# B&R Automation Studio project RobotNewEra (part 11)

#### iolist.c
```c
/************************************************************************************************************************/
/* Object name: iolist.c																								*/
/* Author:      Andreas Hager, B&R																						*/
/* Site:        Eggelsberg                                                                                            	*/
/* Created:     24-Feb-2006                                                                                           	*/
/* Restriction: 													      		                                      	*/
/* Description: Function to read out configured IO data points                                                      	*/
/*----------------------------------------------------------------------------------------------------------------------*/
/* Version 1.00			24-Feb-2006		 Andreas Hager			Official release								  		*/
/*----------------------------------------------------------------------------------------------------------------------*/
/* Version 1.01			13-Dec-2006		 Andreas Hager			Comment added									  		*/
/*----------------------------------------------------------------------------------------------------------------------*/
/* Version 2.00			16-Jul-2008		 Andreas Hager			AS3 - Changes for GCC 4.1.1								*/
/*----------------------------------------------------------------------------------------------------------------------*/
/* Version 2.01			16-Sep-2009		 Andreas Hager			Bugfix for memset in StringParser()						*/
/*----------------------------------------------------------------------------------------------------------------------*/
/* Development tool: B&R Automation Studio V3.0.71.31 SP05 																*/
/*----------------------------------------------------------------------------------------------------------------------*/
/* Comment:                                                                                                           	*/
/************************************************************************************************************************/

#include <ModDiag.h>
#include <bur/plctypes.h>
#include <AsIOMMan.h>
#include <DataObj.h>
#include <string.h>
#include <AsIODiag.h>
#include <Sys_lib.h>
#include <Standard.h>
#include "internal_h.h"

#define	CREATE_HW_INFO		0
#define	ALLOC_MEMORY		1
#define	GET_MODULE_NAME		2
#define	GET_MODULE_PATH		3
#define	CHECK_NEXT_MODULE	4
#define	DISPOSE_INFO		5

#define	MAX_LENGTH			512

#define	PV_NAME_OVERFLOW	50001
#define	FUNCTION_BUSY		65535

static	AsIOMMCopy_typ		IOMapCopy;
static	DatObjDelete_typ	DataModuleDelete;
static	DatObjInfo_typ		DataModuleInfo;

/* Function to get io module information */
unsigned short ModulesInformation(UDINT pModuleInfo);
/* Function to parse iomap data */
unsigned short StringParser(UDINT pBuffer, UDINT pIOData, UDINT pIOCounter, USINT Option);
/* Function to sort io list depending on device */
void SortIOList(UDINT pIOList, UINT IOEntries);

unsigned short IOList(unsigned long pIOInformation)
{	USINT	*Parser = 0, NumberConfiguredModules = 0;
	UINT	xcnt = 0, ycnt  = 0, TotalIOs = 0, OldDigitalInputs = 0, OldDigitalOutputs = 0, OldAnalogInputs = 0, OldAnalogOutputs = 0, DPIndex = 0,
			ModuleStatus = 0, ParserStatus = 0, AllocStatus = 0, StatusFree = 0;
	UDINT	MaxAdr = 0;
	STRING	ParserString[800];

	IODPList_typ			*IOList = 0;
	SingleModuleInfo_typ	*SingleModuleInfo = 0;
	SingleIOEntry_typ		*SingleIOEntry = 0;
	IOStringInfo_typ		EntryInfo;
	IOCounter_typ			IOCounter;
	ModuleInfo_typ			ModuleInformation;

	memset(&(EntryInfo), 0, sizeof(EntryInfo));
	memset(&(ModuleInformation), 0, sizeof(ModuleInformation));
	memset(&(IOCounter), 0, sizeof(IOCounter));

	*(UDINT*)&IOList = pIOInformation;

	/* Get module information */
	do
	{	ModuleStatus = ModulesInformation((UDINT)&(ModuleInformation));
	} while(ModuleStatus == 65535);

	if(ModuleStatus)
	{	return(ModuleStatus);
	}

	/* Number of configured modules */
	NumberConfiguredModules = ModuleInformation.TotalModules - ModuleInformation.IgnoredModules;

	/* Pointer to module information buffer */
	*(UDINT*)&SingleModuleInfo = ModuleInformation.StartAdrBuffer;

	/* Check if io data module already exists */
	DataModuleInfo.enable = 1;
	DataModuleInfo.pName = (UDINT)"iomap_io";
	DatObjInfo(&DataModuleInfo);

	if(DataModuleInfo.status == 0)
	{	DataModuleDelete.enable = 1;
		DataModuleDelete.ident = DataModuleInfo.ident;
		DatObjDelete(&DataModuleDelete);
	}

	/* Generate data module of iomap file */
	do
	{	IOMapCopy.enable = 1;
		IOMapCopy.pModuleName = (UDINT)"iomap";
		IOMapCopy.pNewModule = (UDINT)"iomap_io";
		IOMapCopy.memType = 65;
		AsIOMMCopy(&IOMapCopy);
	} while(IOMapCopy.status == 65535);

	if(IOMapCopy.status)
	{	return(IOMapCopy.status);
	}

	DataModuleInfo.enable = 1;
	DataModuleInfo.pName = (UDINT)"iomap_io";
	DatObjInfo(&DataModuleInfo);

	if(DataModuleInfo.status)
	{	return(DataModuleInfo.status);
	}

	MaxAdr = DataModuleInfo.pDatObjMem + DataModuleInfo.len;

	/* Pointer to the start address of io data module */
	*(UDINT*)&Parser = DataModuleInfo.pDatObjMem;

	while((UDINT)Parser < MaxAdr)
	{
		/* Each line with information starts with <LN */
		if(!memcmp((UDINT*)Parser, "<LN ", 4))
		{	Parser = Parser + 4;

			/* Copy data tiil </LN> */
			for(xcnt = 0; xcnt < 800; xcnt++)
			{	if(!memcmp((UDINT*)Parser, "</LN>", 5))
				{	ParserString[xcnt] = 0;
					Parser = Parser + 5;

					/* Check string for information --> Option = 0 - check number of completed entries */
					ParserStatus = StringParser((UDINT)&(ParserString), (UDINT)&(EntryInfo), (UDINT)&(IOCounter), 0);

					if(ParserStatus)
						return(ParserStatus);

					memset(&(ParserString), 0, sizeof(ParserString));
					break;
				}
				else
				{	ParserString[xcnt] = *Parser;
					Parser++;
				}
			}
		}
		/* Increase pointer */
		else
		{	Parser++;
		}
	}

	TotalIOs = IOCounter.NumberDigitalInputs + IOCounter.NumberDigitalOutputs + IOCounter.NumberAnalogInputs + IOCounter.NumberAnalogOutputs;

	if(TotalIOs == 0)
		return(0);

	/* Allocate memory */
	do
	{	AllocStatus = TMP_alloc(sizeof(SingleIOEntry_typ)*TotalIOs, (void*)&(IOList->StartAdrBuffer));
	} while(AllocStatus == 65535);

	if(AllocStatus)
	{	return(AllocStatus);
	}

	/* Pare data module again */
	memset((void*)IOList->StartAdrBuffer, 0, sizeof(SingleIOEntry_typ)*TotalIOs);
	*(UDINT*)&SingleIOEntry = IOList->StartAdrBuffer;
	memset(&(IOCounter), 0, sizeof(IOCounter));
	memset(&(ParserString), 0, sizeof(ParserString));

	*(UDINT*)&Parser = DataModuleInfo.pDatObjMem;

	while((UDINT)Parser < MaxAdr)
	{
		/* Each line with information starts with <LN */
		if(!memcmp((UDINT*)Parser, "<LN ", 4))
		{	Parser = Parser + 4;

			/* Copy data tiil </LN> */
			for(xcnt = 0; xcnt < 800; xcnt++)
			{	if(!memcmp((UDINT*)Parser, "</LN>", 5))
				{	ParserString[xcnt] = 0;
					Parser = Parser + 5;

					/* Check string for information --> Option = 1 - copy information to EntryInfo */
					ParserStatus = StringParser((UDINT)&(ParserString), (UDINT)&(EntryInfo), (UDINT)&(IOCounter), 1);

					if(ParserStatus)
						return(ParserStatus);

					/* Copy information from EntryInfo to allocated buffer */
					if(OldDigitalInputs != IOCounter.NumberDigitalInputs || OldDigitalOutputs != IOCounter.NumberDigitalOutputs ||
						OldAnalogInputs != IOCounter.NumberAnalogInputs || OldAnalogOutputs != IOCounter.NumberAnalogOutputs)
					{	strcpy((SingleIOEntry + DPIndex)->Device, EntryInfo.Device);
						strcpy((SingleIOEntry + DPIndex)->ID, EntryInfo.ID);
						strcpy((SingleIOEntry + DPIndex)->LogicalName, EntryInfo.LogicalName);
						(SingleIOEntry + DPIndex)->Type = EntryInfo.Type;
						strcpy((SingleIOEntry + DPIndex)->PVName, EntryInfo.PVName);

						memset(&(EntryInfo), 0, sizeof(EntryInfo));

						/* Copy information about io module */
						for(ycnt = 0; ycnt < NumberConfiguredModules; ycnt++)
						{	if(!strcmp((SingleIOEntry + DPIndex)->Device, (SingleModuleInfo + ycnt)->ModulePath))
							{	strcpy((SingleIOEntry + DPIndex)->ModuleName, (SingleModuleInfo + ycnt)->ModuleName);
								break;
							}
						}
						OldDigitalInputs = IOCounter.NumberDigitalInputs;
						OldDigitalOutputs = IOCounter.NumberDigitalOutputs;
						OldAnalogInputs = IOCounter.NumberAnalogInputs;
						OldAnalogOutputs = IOCounter.NumberAnalogOutputs;

						DPIndex++;
					}
					memset(&(ParserString), 0, sizeof(ParserString));
					break;
				}
				else
				{	ParserString[xcnt] = *Parser;
					Parser++;
				}
			}
		}
		else
		{	Parser++;
		}
	}

	/* Free memory with io module information */
	StatusFree = TMP_free(sizeof(SingleModuleInfo_typ)*ModuleInformation.TotalModules, (void*)ModuleInformation.StartAdrBuffer);

	if(StatusFree)
	{	return(StatusFree);
	}

	/* Sort io list */
	SortIOList(IOList->StartAdrBuffer, TotalIOs);

	/* Copy number of ios */
	IOList->NumberDigitalInput = IOCounter.NumberDigitalInputs;
	IOList->NumberDigitalOutput = IOCounter.NumberDigitalOutputs;
	IOList->NumberAnalogInput = IOCounter.NumberAnalogInputs;
	IOList->NumberAnalogOutput = IOCounter.NumberAnalogOutputs;
	IOList->TotalIONumber = IOCounter.NumberDigitalInputs + IOCounter.NumberDigitalOutputs + IOCounter.NumberAnalogInputs + IOCounter.NumberAnalogOutputs;
	return(0);
}

/* Function to get io module information */
unsigned short ModulesInformation(UDINT pModuleInfo)
{	static	DiagCreateInfo_typ		CreateHWInfo;
	static	DiagGetStrInfo_typ		GetModulePath, GetModuleName;
	static	DiagDisposeInfo_typ		DisposeInfo;
	static	SingleModuleInfo_typ	*SingleModuleInfo = 0;

	USINT	*pUSINT1 = 0, *pUSINT2 = 0;
	UINT	Status = 0;
	STRING	ModulePath[40], ModuleName[20];

	ModuleInfo_typ			*ModuleInfo = 0;

	memset(&(ModulePath), 0, sizeof(ModulePath));
	memset(&(ModuleName), 0, sizeof(ModuleName));

	*(UDINT*)&ModuleInfo = pModuleInfo;

	switch(ModuleInfo->Step)
	{
		/* Get information about configured hardware */
		case CREATE_HW_INFO:
			CreateHWInfo.enable = 1;
			CreateHWInfo.infoKind = asdiagCONFIGURED;

			DiagCreateInfo(&CreateHWInfo);
			Status = CreateHWInfo.status;

			if(CreateHWInfo.status == 0)
			{	ModuleInfo->TotalModules = CreateHWInfo.nrEntries;
				ModuleInfo->HWIdent = CreateHWInfo.ident;
				ModuleInfo->Step = ALLOC_MEMORY;
				Status = FUNCTION_BUSY;
			}
		break;

		/* Allocate memory for hardware information depending on number of modules */
		case ALLOC_MEMORY:
			Status = TMP_alloc(sizeof(SingleModuleInfo_typ)*ModuleInfo->TotalModules, (void*)&(ModuleInfo->StartAdrBuffer));

			if(Status == 0)
			{	memset((void*)ModuleInfo->StartAdrBuffer, 0, sizeof(SingleModuleInfo_typ)*ModuleInfo->TotalModules);
				*(UDINT*)&SingleModuleInfo = ModuleInfo->StartAdrBuffer;
				/* Set module index on next module after panel */
				ModuleInfo->ModuleIndex = 1;
				ModuleInfo->IgnoredModules = 1;
				ModuleInfo->Step = GET_MODULE_NAME;
				Status = FUNCTION_BUSY;
			}
		break;

		/* Get name for each hardware module */
		case GET_MODULE_NAME:
			GetModuleName.enable = 1;
			GetModuleName.ident = CreateHWInfo.ident;
			GetModuleName.index = ModuleInfo->ModuleIndex;
			GetModuleName.infoCode = asdiagCONFIG_MODULE;
			GetModuleName.pBuffer = (UDINT)ModuleName;
			GetModuleName.bufferLen = sizeof(ModuleName);

			DiagGetStrInfo(&GetModuleName);
			Status = GetModuleName.status;

			if(GetModuleName.status == 0)
			{	*(UDINT*)&pUSINT1 = (UDINT)(ModuleName + 1);
				*(UDINT*)&pUSINT2 = (UDINT)(ModuleName + 2);

				/* Ignore IF and ACxxx */
				if((*pUSINT1 == 'I' && *pUSINT2 == 'F') || (*pUSINT1 == 'A' && *pUSINT2 == 'C'))
				{	ModuleInfo->IgnoredModules++;
					ModuleInfo->Step = CHECK_NEXT_MODULE;
				}
				else
				{	strcpy((SingleModuleInfo + (ModuleInfo->ModuleIndex - ModuleInfo->IgnoredModules))->ModuleName, ModuleName);
					ModuleInfo->Step = GET_MODULE_PATH;
				}
				Status = FUNCTION_BUSY;
			}
		break;

		/* Get path for each hardware module */
		case GET_MODULE_PATH:
			GetModulePath.enable = 1;
			GetModulePath.ident = CreateHWInfo.ident;
			GetModulePath.index = ModuleInfo->ModuleIndex;
			GetModulePath.infoCode = asdiagPATH;
			GetModulePath.pBuffer = (UDINT)ModulePath;
			GetModulePath.bufferLen = sizeof(ModulePath);

			DiagGetStrInfo(&GetModulePath);
			Status = GetModulePath.status;

			if(GetModulePath.status == 0)
			{	strcpy((SingleModuleInfo + (ModuleInfo->ModuleIndex - ModuleInfo->IgnoredModules))->ModulePath, ModulePath);
				ModuleInfo->Step = CHECK_NEXT_MODULE;
				Status = FUNCTION_BUSY;
			}
		break;

		/* Select nex module */
		case CHECK_NEXT_MODULE:
			if(ModuleInfo->ModuleIndex < ModuleInfo->TotalModules - 1)
			{	ModuleInfo->ModuleIndex++;
				ModuleInfo->Step = GET_MODULE_NAME;
			}
			else
			{	ModuleInfo->Step = DISPOSE_INFO;
			}
			Status = FUNCTION_BUSY;
		break;

		/* Dispose information */
		case DISPOSE_INFO:
			DisposeInfo.enable = 1;
			DisposeInfo.ident = ModuleInfo->HWIdent;

			DiagDisposeInfo(&DisposeInfo);

			if(DisposeInfo.status == 0)
			{	ModuleInfo->Step = CREATE_HW_INFO;
			}
		break;
	}
	return(Status);
}

/* Function to parse iomap data */
unsigned short StringParser(UDINT pBuffer, UDINT pIOData, UDINT pIOCounter, USINT Option)
{	USINT	*Parser = 0, Element = 0;
	UINT xcnt = 0;
	STRING	Data[MAX_LENGTH], ID[60], Type[40], DType[40], Device1[60], DPName1[34], Kind1[40], Device2[60], DPName2[34], Kind2[40];

	IOStringInfo_typ	*EntryInfo = 0;
	IOCounter_typ		*IOCounter = 0;

	memset(&(Data), 0, sizeof(Data));
	memset(&(ID), 0, sizeof(ID));
	memset(&(Type), 0, sizeof(Type));
	memset(&(DType), 0, sizeof(DType));
	memset(&(Device1), 0, sizeof(Device1));
	memset(&(DPName1), 0, sizeof(DPName1));
	memset(&(Kind1), 0, sizeof(Kind1));
	memset(&(Device2), 0, sizeof(Device2));
	memset(&(DPName2), 0, sizeof(DPName2));
	memset(&(Kind2), 0, sizeof(Kind2));

	*(UDINT*)&Parser = pBuffer;
	*(UDINT*)&EntryInfo = pIOData;
	*(UDINT*)&IOCounter = pIOCounter;

	while(*Parser)
	{	/* Information starts with " */
		while(*Parser != '"' && *Parser)
		{	Parser++;
		}
		if(!*Parser)
			break;
		else
			Parser++;

		/* Information ends with " */
		while(*Parser != '"' && *Parser)
		{	Data[xcnt] = *Parser;
			Parser++;
			xcnt++;
			if(xcnt == MAX_LENGTH)
				return(PV_NAME_OVERFLOW);
		}
		Parser++;
		Data[xcnt] = 0;
		xcnt = 0;

		/* Element 0 --> IO ID */
		if(Element == 0)
		{	strcpy(ID, Data);
			memcpy(Type, Data, 3);
		}
		/* Element 1 --> Data type */
		else if(Element == 1)
		{	strcpy(DType, Data);
		}
		/* Element 2 --> Device */
		else if(Element == 2)
		{	strcpy(Device1, Data);
		}
		/* Element 3 --> Data point name */
		else if(Element == 3)
		{	strcpy(DPName1, Data);
		}
		/* Element 4 --> Kind */
		else if(Element == 4)
		{	strcpy(Kind1, Data);
		}
		/* Element 5 --> Device */
		else if(Element == 5)
		{	strcpy(Device2, Data);
		}
		/* Element 6 --> Data point name */
		else if(Element == 6)
		{	strcpy(DPName2, Data);
		}
		/* Elemtn 7 --> Kind */
		else if(Element == 7)
		{	strcpy(Kind2, Data);
		}

		Element++;
		memset(&(Data), 0, sizeof(Data));
	}

	/* If less than 8 elements are detected --> information is completed */
	if(Element != 8)
	{	Element = 0;
		return(0);
	}

	/* Type %IX --> Digital input */
	if(Element == 8 && !strcmp(Type, "%IX"))
	{	IOCounter->NumberDigitalInputs++;
	}
	/* Type %QX --> Digital output */
	else if(Element == 8 && !strcmp(Type, "%QX"))
	{	IOCounter->NumberDigitalOutputs++;
	}
	/* Type %IW --> Analog input */
	else if(Element == 8 && !strcmp(Type, "%IW"))
	{	IOCounter->NumberAnalogInputs++;
	}
	/* Type %QW --> Analog output */
	else if(Element == 8 && !strcmp(Type, "%QW"))
	{	IOCounter->NumberAnalogOutputs++;
	}

	/* If option = 1 --> copy all information to EntryInfo */
	if(Option == 1 && Element == 8)
	{	strcpy(EntryInfo->ID, ID);

		if(!strcmp(Type, "%IX"))
		{	EntryInfo->Type = 1;
			if(!strcmp(Kind1, "io"))
			{	strcpy(EntryInfo->LogicalName, DPName1);
			}
			else if(!strcmp(Kind2, "io"))
			{	strcpy(EntryInfo->LogicalName, DPName2);
			}
		}
		else if(!strcmp(Type, "%QX"))
		{	EntryInfo->Type = 2;
			if(!strcmp(Kind1, "io"))
			{	strcpy(EntryInfo->LogicalName, DPName1);
			}
			else if(!strcmp(Kind2, "io"))
			{	strcpy(EntryInfo->LogicalName, DPName2);
			}
		}
		else if(!strcmp(Type, "%IW"))
		{	EntryInfo->Type = 3;
			if(!strcmp(Kind1, "io"))
			{	strcpy(EntryInfo->LogicalName, DPName1);
			}
			else if(!strcmp(Kind2, "io"))
			{	strcpy(EntryInfo->LogicalName, DPName2);
			}
		}
		else if(!strcmp(Type, "%QW"))
		{	EntryInfo->Type = 4;
			if(!strcmp(Kind1, "io"))
			{	strcpy(EntryInfo->LogicalName, DPName1);
			}
			else if(!strcmp(Kind2, "io"))
			{	strcpy(EntryInfo->LogicalName, DPName2);
			}
		}

		if(!strcmp(Kind1, "pv"))
		{	strcpy(EntryInfo->PVName, DPName1);
			strcpy(EntryInfo->Device, Device2);
		}
		else if(!strcmp(Kind2, "pv"))
		{	strcpy(EntryInfo->PVName, DPName2);
			strcpy(EntryInfo->Device, Device1);
		}
	}

	Element = 0;
	return(0);
}

/* Function to sort io list depending on device */
void SortIOList(UDINT pIOList, UINT IOEntries)
{	STRING				ParserString1[60], ParserString2[60], *Parser1, *Parser2;
	UINT				IOType = 0, xcnt = 0, ycnt = 0, zcnt = 0, ExchangeData;
	DINT				Result = 0;
	SingleIOEntry_typ	*SingleIOEntry = 0;
	SingleIOEntry_typ	IOEntryData;

	memset(&(ParserString1), 0, sizeof(ParserString1));
	memset(&(ParserString2), 0, sizeof(ParserString2));
	memset(&(IOEntryData), 0, sizeof(IOEntryData));

	*(UDINT*)&SingleIOEntry = pIOList;

	for(xcnt = 0; xcnt < IOEntries - 1; xcnt++)
	{	for(ycnt = 0; ycnt < IOEntries - 1 - xcnt; ycnt++)
		{	/* Pointer to io ID of entry */
			*(UDINT*)&Parser1 = (UDINT)(SingleIOEntry + ycnt)->ID;
			/* Pointer to io ID of the next entry */
			*(UDINT*)&Parser2 = (UDINT)(SingleIOEntry + ycnt + 1)->ID;

			while(*Parser1 && *Parser2)
			{	while(*Parser1 != '.' && *Parser2 != '.' && IOType == 0)
				{	Parser1++;
					Parser2++;
				}
				if(IOType == 0)
				{	Parser1++;
					Parser2++;
					IOType = 1;
				}

				while(*Parser1 != '.' && *Parser1)
				{	ParserString1[zcnt] = *Parser1;
					Parser1++;
					zcnt++;
				}
				Parser1++;
				ParserString1[zcnt] = 0;
				zcnt = 0;

				while(*Parser2 != '.' && *Parser2)
				{	ParserString2[zcnt] = *Parser2;
					Parser2++;
					zcnt++;
				}
				Parser2++;
				ParserString2[zcnt] = 0;
				zcnt = 0;

				Result = strcmp(ParserString1, ParserString2);

				if(Result < 0)
				{	break;
				}
				else if(Result > 0 && memcmp(ParserString1, "ModuleOk", 8) && memcmp(ParserString1, "SerialNumber", 12) && memcmp(ParserString1, "ModuleID", 8) &&
					memcmp(ParserString1, "HardwareVariant", 15) && memcmp(ParserString1, "FirmwareVersion", 15))
				{	ExchangeData = 1;
					break;
				}
			}

			/* Exchange data */
			if(ExchangeData == 1)
			{	memcpy(&(IOEntryData), (SingleIOEntry + ycnt), sizeof(IOEntryData));
				memcpy((SingleIOEntry + ycnt), (SingleIOEntry + ycnt + 1), sizeof(IOEntryData));
				memcpy((SingleIOEntry + ycnt + 1), &(IOEntryData), sizeof(IOEntryData));

				ExchangeData = 0;
			}
			memset(&(ParserString1), 0, sizeof(ParserString1));
			memset(&(ParserString2), 0, sizeof(ParserString2));
			memset(&(IOEntryData), 0, sizeof(IOEntryData));
			IOType = 0;
		}
	}
}
```

#### iostatus.c
```c
/************************************************************************************************************************/
/* Object name: iostatus.c																								*/
/* Author:      Andreas Hager, B&R																						*/
/* Site:        Eggelsberg                                                                                            	*/
/* Created:     24-Feb-2006                                                                                           	*/
/* Restriction: 													      		                                      	*/
/* Description: Function to handle configured IO data points	                                                      	*/
/*----------------------------------------------------------------------------------------------------------------------*/
/* Version 1.00			24-Feb-2006		 Andreas Hager			Official release								  		*/
/*----------------------------------------------------------------------------------------------------------------------*/
/* Version 1.01			12-Dec-2006		 Andreas Hager			More IOs can be handled and commment added 		  		*/
/*----------------------------------------------------------------------------------------------------------------------*/
/* Version 2.00			16-Jul-2008		 Andreas Hager			AS3 - Changes for GCC 4.1.1								*/
/*----------------------------------------------------------------------------------------------------------------------*/
/* Development tool: B&R Automation Studio V3.0.71.10 																  	*/
/*----------------------------------------------------------------------------------------------------------------------*/
/* Comment:                                                                                                           	*/
/************************************************************************************************************************/

#include <ModDiag.h>
#include <bur/plctypes.h>
#include <AsIOMMan.h>
#include <DataObj.h>
#include <string.h>
#include <AsIO.h>
#include <AsIODiag.h>
#include <Sys_lib.h>
#include "internal_h.h"

#define	FORCE_STATUS	0x04

#define	CHECK_DP_ACTIONS	0
#define	ENABLE_FORCE		1
#define	SET_FORCE_VALUE		2
#define	GET_DP_STATUS		3
#define	DISABLE_FORCE		4
#define	NEXT_DP				5

#define	FUNCTION_BUSY	65535

static	AsIODPStatus_typ		IODPStatus;
static	AsIOEnableForcing_typ	IODPEnableForce;
static	AsIODisableForcing_typ	IODPDisableForce;
static	AsIOSetForceValue_typ	IODPSetForceValue;

unsigned short IOStatus(unsigned long pIOList, unsigned long pStatusBuffer, unsigned short Elements, unsigned long pEnableForce, unsigned long pForceValue)
{	static	USINT		Step = 0;
	static	UINT		DPIndex = 0;

	USINT	StatusFlag = 0, ForceStatus = 0;
	UINT	Status = 0;

	SingleIOEntry_typ		*SingleIOEntry = 0;
	SingleIOStatus_typ		*SingleIOStatus = 0;
	BOOL					*EnableForce = 0;
	DINT					*ForceValue = 0;

	*(UDINT*)&SingleIOEntry = pIOList;
	*(UDINT*)&SingleIOStatus = pStatusBuffer;
	*(UDINT*)&EnableForce = pEnableForce;
	*(UDINT*)&ForceValue = pForceValue;

	if(Elements <= 0)
	{	return(0);
	}

	switch(Step)
	{	/* Check actions for data point */
		case CHECK_DP_ACTIONS:
			/* Force data point - forcing data point */
			if(*(EnableForce + DPIndex) == 1)
			{	if((SingleIOStatus + DPIndex)->ForceActive == 0)
				{	/* Call funtion block to enable forcing */
					IODPEnableForce.enable = 1;
					IODPEnableForce.pDatapoint = (UDINT)(SingleIOEntry + DPIndex)->ID;

					AsIOEnableForcing(&(IODPEnableForce));
					Status = IODPEnableForce.status;

					if(IODPEnableForce.status == 0)
					{	Status = FUNCTION_BUSY;
						Step = SET_FORCE_VALUE;
					}
				}
				else
				{	Status = FUNCTION_BUSY;
					Step = SET_FORCE_VALUE;
				}
			}
			else
			{	Status = FUNCTION_BUSY;
				Step = GET_DP_STATUS;
			}
		break;

		/* Set force value for data point */
		case SET_FORCE_VALUE:
			/* Call function block to set force value */
			IODPSetForceValue.enable = 1;
			IODPSetForceValue.pDatapoint = (UDINT)(SingleIOEntry + DPIndex)->ID;
			/* Force value */
			IODPSetForceValue.value = *(ForceValue + DPIndex);

			AsIOSetForceValue(&(IODPSetForceValue));
			Status = IODPSetForceValue.status;

			if(IODPSetForceValue.status == 0)
			{	Status = FUNCTION_BUSY;
				Step = GET_DP_STATUS;
			}
		break;

		/* Get data point status */
		case GET_DP_STATUS:
			/* Call functio block to get data point status */
			IODPStatus.enable = 1;
			IODPStatus.pDatapoint = (UDINT)(SingleIOEntry + DPIndex)->ID;

			AsIODPStatus(&(IODPStatus));
			Status = IODPStatus.status;

			if(IODPStatus.status == 0)
			{	/* Copy data to io status buffer */
				(SingleIOStatus + DPIndex)->ActValue = (DINT)IODPStatus.value;
				(SingleIOStatus + DPIndex)->ActForceValue = (DINT)IODPStatus.forceValue;
				(SingleIOStatus + DPIndex)->DataType = IODPStatus.datatype;

				StatusFlag = IODPStatus.flags;
				ForceStatus = IODPStatus.flags & FORCE_STATUS;

				if(StatusFlag==39 || StatusFlag == 23 )
				{
					(SingleIOStatus + DPIndex)->ActValue = (DINT)IODPStatus.forceValue;
				}

				if(ForceStatus == 4)
				{	(SingleIOStatus + DPIndex)->ForceActive = 1;
				}
				else
				{	(SingleIOStatus + DPIndex)->ForceActive = 0;
				}

				Status = FUNCTION_BUSY;
				Step = DISABLE_FORCE;
			}
		break;

		/* Disable forcing */
		case DISABLE_FORCE:
			/* Forcing data point */
			if(*(EnableForce + DPIndex) == 0 && (SingleIOStatus + DPIndex)->ForceActive == 1)
			{	/* Call function block to disable forcing */
				IODPDisableForce.enable = 1;
				IODPDisableForce.pDatapoint = (UDINT)(SingleIOEntry + DPIndex)->ID;

				AsIODisableForcing(&(IODPDisableForce));
				Status = IODPDisableForce.status;

				if(IODPDisableForce.status == 0)
				{	Status = FUNCTION_BUSY;
					Step = NEXT_DP;
				}
			}
			else
			{	Status = FUNCTION_BUSY;
				Step = NEXT_DP;
			}
		break;

		/* Select next io data point */
		case NEXT_DP:
			if(DPIndex < Elements - 1)
			{	DPIndex++;
				Status = FUNCTION_BUSY;
				Step = CHECK_DP_ACTIONS;
			}
			else
			{	DPIndex = 0;
				Status = 0;
				Step = CHECK_DP_ACTIONS;
			}
		break;
	}
	return(Status);
}
```

#### modulediagnose.c
```c
/************************************************************************************************************************/
/* Object name: modulediagnose.c																						*/
/* Author:      Andreas Hager, B&R																						*/
/* Site:        Eggelsberg                                                                                            	*/
/* Created:     20-Dec-2005                                                                                           	*/
/* Restriction: 													      		                                      	*/
/* Description: Function-block for module-diagnose with alarmbits                                                      	*/
/*----------------------------------------------------------------------------------------------------------------------*/
/* Version 1.00			20-Dec-2005		 Andreas Hager			Official release								  		*/
/*----------------------------------------------------------------------------------------------------------------------*/
/* Version 1.01			03-Feb-2006		 Andreas Hager			Changed module name for "module is only configured" 	*/
/*																from empty to "ModuleName"								*/
/*----------------------------------------------------------------------------------------------------------------------*/
/* Version 1.02			21-Apr-2006		 Andreas Hager			Problem with waiting-timer fixed and Buffer-overflow	*/
/*----------------------------------------------------------------------------------------------------------------------*/
/* Version 2.00			16-Jul-2008		 Andreas Hager			AS3 - Changes for GCC 4.1.1								*/
/*----------------------------------------------------------------------------------------------------------------------*/
/* Development tool: B&R Automation Studio V3.0.71.10																  	*/
/*----------------------------------------------------------------------------------------------------------------------*/
/* Comment:                                                                                                           	*/
/************************************************************************************************************************/

#include <ModDiag.h>
#include <bur/plctypes.h>
#include <AsIODiag.h>
#include <string.h>
#include <Standard.h>

#define	CREATE_HW_INFO				0
#define	CHECK_MODULESTATE			1
#define	CHECK_CONNECTED				2
#define	GET_CONFIGUREDMODULE		3
#define	GET_MODULEPATH				4
#define	CHECK_OLD_MODULE_PATH		5
#define	RESET_MODULE_ALARMS1		6
#define	CHECK_OLD_MODULE_ALARMS		7
#define	RESET_MODULE_ALARMS2		8
#define	CHECK_NEW_ALARMMESSAGES		9
#define	SET_ALARMMESSAGES			10
#define	CHECK_NEXT_MODULE			11
#define	CHECK_MODULENUMBER			12
#define	CHECK_NOT_NEEDED_ALARMS		13
#define	RESET_NOT_NEEDED_ALARMS		14
#define	CHECK_RESET_NEXT_MODULE		15
#define	DISPOSE_INFO				16
#define	WAIT						17

#define	MODULE_ONLY_CONFIGURED	1
#define	MODULE_ONLY_INSERTED	2
#define	MODULE_OK				3
#define	VAR_MODULE_PLUGGED		4

#define	OFFSET_MODULE_ONLY_CONFIGURED	0
#define	OFFSET_MODULE_ONLY_INSERTED		100
#define	OFFSET_VARIOUS_MODULE_PLUGGED	200

#define	WRONG_OPTION_SELECTED	50000
#define	FUNCTION_BUSY			65535

static	DiagCreateInfo_typ	CreateHWInfo;
static	DiagGetStrInfo_typ	GetModuleName, GetModulePath;
static	DiagGetNumInfo_typ	GetModuleState;
static	DiagDisposeInfo_typ	DisposeInfo;
/*static	TON_typ				WaitTimer;*/

void ModuleDiagnose(ModuleDiagnose_typ* pModuleInfo)
{	ModuleInformationBuffer_typ	*ModuleInfoBuffer;
	ModuleAlarmInformation_typ	*ModuleAlarmInfo;

	USINT	*pUSINT1 = 0, *pUSINT2 = 0;
	STRING	ModuleName[40], ModulePath[40];
	DINT	PathResult = 0;
	BOOL	AlarmMessage = 0;

	memset(&ModuleName, 0, sizeof(ModuleName));
	memset(&ModulePath, 0, sizeof(ModulePath));

	*(UDINT*)&ModuleInfoBuffer = pModuleInfo->AdrModuleInformationBuffer;
	*(UDINT*)&ModuleAlarmInfo = pModuleInfo->AdrAlarmInformation;

	if(pModuleInfo->Option > 3)
	{	pModuleInfo->status = WRONG_OPTION_SELECTED;
		return;
	}

	switch(pModuleInfo->Step)
	{
		/* create the information about configured and plugged hardware */
		case CREATE_HW_INFO:
			pModuleInfo->status = FUNCTION_BUSY;

			CreateHWInfo.enable = 1;
			CreateHWInfo.infoKind = asdiagALL;

			DiagCreateInfo(&CreateHWInfo);

			if(CreateHWInfo.status == 0)
			{	pModuleInfo->NumberNotCheckedModules = 0;
				pModuleInfo->NumberOfTotalModules = CreateHWInfo.nrEntries;

				/* check option if panel and if information is requested */
				/* Option 0 ==> All hardware 				*/
				/* Option 1 ==> Without panel and IF		*/
				/* Option 2 ==> Without AC					*/
				/* Option 3 ==> Without panel, IF and AC	*/
				if(pModuleInfo->Option == 0 || pModuleInfo->Option == 2)
				{	pModuleInfo->ModuleIndex = 0;
				}
				else if(pModuleInfo->Option == 1 || pModuleInfo->Option == 3)
				{	pModuleInfo->NumberNotCheckedModules++;
					pModuleInfo->ModuleIndex = 1;
				}

				pModuleInfo->Step = CHECK_MODULESTATE;
			}
			else if(CreateHWInfo.status != 65535)
			{	pModuleInfo->status = CreateHWInfo.status;
				return;
			}
		break;

		/* check state of module */
		case CHECK_MODULESTATE:
			GetModuleState.enable = 1;
			GetModuleState.ident = CreateHWInfo.ident;
			GetModuleState.index = pModuleInfo->ModuleIndex;
			GetModuleState.infoCode = asdiagMODUL_STATE;

			DiagGetNumInfo(&GetModuleState);

			if(GetModuleState.status == 0)
			{	pModuleInfo->ActualModuleInformation.ModuleState = GetModuleState.value;
				pModuleInfo->Step = CHECK_CONNECTED;
			}
			else if(GetModuleState.status != 65535)
			{	pModuleInfo->status = GetModuleState.status;
				return;
			}
		break;

		/* get module-name and handle module-data */
		case CHECK_CONNECTED:
			if(GetModuleState.value == MODULE_ONLY_CONFIGURED || GetModuleState.value == MODULE_OK)
			{	GetModuleName.infoCode = asdiagCONFIG_MODULE;
			}
			else if(GetModuleState.value == MODULE_ONLY_INSERTED || GetModuleState.value == VAR_MODULE_PLUGGED)
			{	GetModuleName.infoCode = asdiagPLUGGED_MODULE;
			}

			GetModuleName.enable = 1;
			GetModuleName.ident = CreateHWInfo.ident;
			GetModuleName.index = pModuleInfo->ModuleIndex;
			GetModuleName.pBuffer = (UDINT)ModuleName;
			GetModuleName.bufferLen = sizeof(ModuleName);

			DiagGetStrInfo(&GetModuleName);

			if(GetModuleName.status == 0)
			{	*(UDINT*)&pUSINT1 = (UDINT)(ModuleName + 1);
				*(UDINT*)&pUSINT2 = (UDINT)(ModuleName + 2);

				if((*pUSINT1 == 'I' && *pUSINT2 == 'F') && pModuleInfo->Option == 1)
				{	pModuleInfo->NumberNotCheckedModules++;
					pModuleInfo->Step = CHECK_NEXT_MODULE;
				}

				else if((*pUSINT1 == 'A' && *pUSINT2 == 'C') && pModuleInfo->Option == 2)
				{	pModuleInfo->NumberNotCheckedModules++;
					pModuleInfo->Step = CHECK_NEXT_MODULE;
				}
				else if(((*pUSINT1 == 'I' && *pUSINT2 == 'F') || (*pUSINT1 == 'A' && *pUSINT2 == 'C')) && pModuleInfo->Option == 3)
				{	pModuleInfo->NumberNotCheckedModules++;
					pModuleInfo->Step = CHECK_NEXT_MODULE;
				}
				else
				{	/* module is only configured --> module is missing */
					if(pModuleInfo->ActualModuleInformation.ModuleState == MODULE_ONLY_CONFIGURED)
					{	/* copy moduledata */
						pModuleInfo->ActualModuleInformation.ModuleState = MODULE_ONLY_CONFIGURED;
						pModuleInfo->ActualModuleInformation.ModuleColor = 51;
						strcpy(pModuleInfo->ActualModuleInformation.ModuleName, ModuleName);
						strcpy(pModuleInfo->ActualModuleInformation.ErrorModuleName, ModuleName);

						/* get module-path */
						pModuleInfo->Step = GET_MODULEPATH;
					}
					/* module is only inserted --> module is not configured */
					else if(pModuleInfo->ActualModuleInformation.ModuleState == MODULE_ONLY_INSERTED)
					{	/* copy moduledata */
						pModuleInfo->ActualModuleInformation.ModuleState = MODULE_ONLY_INSERTED;
						pModuleInfo->ActualModuleInformation.ModuleColor = 46;
						strcpy(pModuleInfo->ActualModuleInformation.ModuleName, ModuleName);

						/* get module-path */
						pModuleInfo->Step = GET_MODULEPATH;
					}
					/* modulestate is OK */
					else if(pModuleInfo->ActualModuleInformation.ModuleState == MODULE_OK)
					{	/* copy moduledata */
						pModuleInfo->ActualModuleInformation.ModuleState = MODULE_OK;
						pModuleInfo->ActualModuleInformation.ModuleColor = 226;
						strcpy(pModuleInfo->ActualModuleInformation.ModuleName, ModuleName);

						/* get module-path */
						pModuleInfo->Step = GET_MODULEPATH;
					}
					/* various module is plugged */
					else if(pModuleInfo->ActualModuleInformation.ModuleState == VAR_MODULE_PLUGGED)
					{	/* copy moduledata */
						pModuleInfo->ActualModuleInformation.ModuleState = VAR_MODULE_PLUGGED;
						pModuleInfo->ActualModuleInformation.ModuleColor = 51;
						strcpy(pModuleInfo->ActualModuleInformation.ModuleName, ModuleName);

						/* get information about configured module */
						pModuleInfo->Step = GET_CONFIGUREDMODULE;
					}
				}
			}
			else if(GetModuleName.status != 65535)
			{	pModuleInfo->status = GetModuleName.status;
				return;
			}
		break;

		/* if various module is plugged, get information about configured module */
		case GET_CONFIGUREDMODULE:
			GetModuleName.enable = 1;
			GetModuleName.ident = CreateHWInfo.ident;
			GetModuleName.index = pModuleInfo->ModuleIndex;
			GetModuleName.infoCode = asdiagCONFIG_MODULE;
			GetModuleName.pBuffer = (UDINT)ModuleName;
			GetModuleName.bufferLen = sizeof(ModuleName);

			DiagGetStrInfo(&GetModuleName);

			if(GetModuleName.status == 0)
			{	/* copy moduledata */
				strcpy(pModuleInfo->ActualModuleInformation.ErrorModuleName, ModuleName);

				/* get module-path */
				pModuleInfo->Step = GET_MODULEPATH;
			}
			else if(GetModuleName.status != 65535)
			{	pModuleInfo->status = GetModuleName.status;
				return;
			}
		break;

		/* get module-path */
		case GET_MODULEPATH:
			GetModulePath.enable = 1;
			GetModulePath.ident = CreateHWInfo.ident;
			GetModulePath.index = pModuleInfo->ModuleIndex;
			GetModulePath.infoCode = asdiagPATH;
			GetModulePath.pBuffer = (UDINT)ModulePath;
			GetModulePath.bufferLen = sizeof(ModulePath);

			DiagGetStrInfo(&GetModulePath);

			if(GetModulePath.status == 0)
			{	strcpy(pModuleInfo->ActualModuleInformation.ModulePath, ModulePath);
				pModuleInfo->Step = CHECK_OLD_MODULE_PATH;
			}
			else if(GetModulePath.status != 65535)
			{	pModuleInfo->status = GetModulePath.status;
				return;
			}
		break;

		/* check old module path */
		case CHECK_OLD_MODULE_PATH:
			/* compare actual and old path of module */
			PathResult = strcmp(pModuleInfo->ActualModuleInformation.ModulePath, pModuleInfo->PathBuffer[pModuleInfo->ModuleNumber]);

			if(PathResult != 0)
			{	if(ModuleAlarmInfo->AlarmBitField[pModuleInfo->ModuleNumber + OFFSET_MODULE_ONLY_CONFIGURED] == 1)
				{	/* copy information for textsnippets */
					strcpy(ModuleAlarmInfo->ErrorModulePath, ModuleInfoBuffer->ModuleInformation[pModuleInfo->ModuleNumber].ModulePath);
					strcpy(ModuleAlarmInfo->ErrorModuleName, ModuleInfoBuffer->ModuleInformation[pModuleInfo->ModuleNumber].ErrorModuleName);
					AlarmMessage = 1;
				}
				else if(ModuleAlarmInfo->AlarmBitField[pModuleInfo->ModuleNumber + OFFSET_MODULE_ONLY_INSERTED] == 1)
				{	/* copy information for textsnippets */
					strcpy(ModuleAlarmInfo->ErrorModulePath, ModuleInfoBuffer->ModuleInformation[pModuleInfo->ModuleNumber].ModulePath);
					strcpy(ModuleAlarmInfo->ErrorModuleName, ModuleInfoBuffer->ModuleInformation[pModuleInfo->ModuleNumber].ModuleName);
					AlarmMessage = 1;
				}
				else if(ModuleAlarmInfo->AlarmBitField[pModuleInfo->ModuleNumber + OFFSET_VARIOUS_MODULE_PLUGGED] == 1)
				{	/* copy information for textsnippets */
					strcpy(ModuleAlarmInfo->ErrorModulePath, ModuleInfoBuffer->ModuleInformation[pModuleInfo->ModuleNumber].ModulePath);
					strcpy(ModuleAlarmInfo->ErrorModuleName, ModuleInfoBuffer->ModuleInformation[pModuleInfo->ModuleNumber].ErrorModuleName);
					AlarmMessage = 1;
				}
			}

			strcpy(pModuleInfo->PathBuffer[pModuleInfo->ModuleNumber], pModuleInfo->ActualModuleInformation.ModulePath);

			/* reset other alarmmessages */
			if(AlarmMessage == 0)
			{	pModuleInfo->Step = CHECK_OLD_MODULE_ALARMS;
			}
			else
			{	AlarmMessage = 0;
				pModuleInfo->LastStep = CHECK_OLD_MODULE_PATH;
				pModuleInfo->Step = WAIT;
			}
		break;

		/* reset module alarms */
		case RESET_MODULE_ALARMS1:
			if(ModuleAlarmInfo->AlarmBitField[pModuleInfo->ModuleNumber + OFFSET_MODULE_ONLY_CONFIGURED] == 1)
			{	/* reset alarm */
				ModuleAlarmInfo->AlarmBitField[pModuleInfo->ModuleNumber + OFFSET_MODULE_ONLY_CONFIGURED] = 0;
			}
			else if(ModuleAlarmInfo->AlarmBitField[pModuleInfo->ModuleNumber + OFFSET_MODULE_ONLY_INSERTED] == 1)
			{	/* reset alarm */
				ModuleAlarmInfo->AlarmBitField[pModuleInfo->ModuleNumber + OFFSET_MODULE_ONLY_INSERTED] = 0;
			}
			else if(ModuleAlarmInfo->AlarmBitField[pModuleInfo->ModuleNumber + OFFSET_VARIOUS_MODULE_PLUGGED] == 1)
			{	/* reset alarm */
				ModuleAlarmInfo->AlarmBitField[pModuleInfo->ModuleNumber + OFFSET_VARIOUS_MODULE_PLUGGED] = 0;
			}
			pModuleInfo->LastStep = RESET_MODULE_ALARMS1;
			pModuleInfo->Step = WAIT;
		break;

		/* check old module alarms */
		case CHECK_OLD_MODULE_ALARMS:

			if(pModuleInfo->ActualModuleInformation.ModuleState == MODULE_ONLY_CONFIGURED)
			{	/* reset other alarmbits */
				if(ModuleAlarmInfo->AlarmBitField[pModuleInfo->ModuleNumber + OFFSET_MODULE_ONLY_INSERTED] == 1)
				{	/* copy information for textsnippets */
					strcpy(ModuleAlarmInfo->ErrorModulePath, ModuleInfoBuffer->ModuleInformation[pModuleInfo->ModuleNumber].ModulePath);
					strcpy(ModuleAlarmInfo->ErrorModuleName, ModuleInfoBuffer->ModuleInformation[pModuleInfo->ModuleNumber].ModuleName);
					AlarmMessage = 1;
				}
				else if(ModuleAlarmInfo->AlarmBitField[pModuleInfo->ModuleNumber + OFFSET_VARIOUS_MODULE_PLUGGED] == 1)
				{	/* copy information for textsnippets */
					strcpy(ModuleAlarmInfo->ErrorModulePath, ModuleInfoBuffer->ModuleInformation[pModuleInfo->ModuleNumber].ModulePath);
					strcpy(ModuleAlarmInfo->ErrorModuleName, ModuleInfoBuffer->ModuleInformation[pModuleInfo->ModuleNumber].ErrorModuleName);
					AlarmMessage = 1;
				}
			}
			/* module is only inserted --> module only inserted */
			else if(pModuleInfo->ActualModuleInformation.ModuleState == MODULE_ONLY_INSERTED)
			{	/* reset other alarmbits */
				if(ModuleAlarmInfo->AlarmBitField[pModuleInfo->ModuleNumber + OFFSET_MODULE_ONLY_CONFIGURED] == 1)
				{	/* copy information for textsnippets */
					strcpy(ModuleAlarmInfo->ErrorModulePath, ModuleInfoBuffer->ModuleInformation[pModuleInfo->ModuleNumber].ModulePath);
					strcpy(ModuleAlarmInfo->ErrorModuleName, ModuleInfoBuffer->ModuleInformation[pModuleInfo->ModuleNumber].ErrorModuleName);
					AlarmMessage = 1;
				}
				else if(ModuleAlarmInfo->AlarmBitField[pModuleInfo->ModuleNumber + OFFSET_VARIOUS_MODULE_PLUGGED] == 1)
				{	/* copy information for textsnippets */
					strcpy(ModuleAlarmInfo->ErrorModulePath, ModuleInfoBuffer->ModuleInformation[pModuleInfo->ModuleNumber].ModulePath);
					strcpy(ModuleAlarmInfo->ErrorModuleName, ModuleInfoBuffer->ModuleInformation[pModuleInfo->ModuleNumber].ErrorModuleName);
					AlarmMessage = 1;
				}
			}
			/* modulestate is OK */
			else if(pModuleInfo->ActualModuleInformation.ModuleState == MODULE_OK)
			{	/* if module-only-configured alarmbit is set --> reset */
				if(ModuleAlarmInfo->AlarmBitField[pModuleInfo->ModuleNumber + OFFSET_MODULE_ONLY_CONFIGURED] == 1)
				{	/* copy information for textsnippets */
					strcpy(ModuleAlarmInfo->ErrorModulePath, ModuleInfoBuffer->ModuleInformation[pModuleInfo->ModuleNumber].ModulePath);
					strcpy(ModuleAlarmInfo->ErrorModuleName, ModuleInfoBuffer->ModuleInformation[pModuleInfo->ModuleNumber].ErrorModuleName);
					AlarmMessage = 1;
				}
				/* if module-only-inserted alarmbit is set --> reset */
				else if(ModuleAlarmInfo->AlarmBitField[pModuleInfo->ModuleNumber + OFFSET_MODULE_ONLY_INSERTED] == 1)
				{	/* copy information for textsnippets */
					strcpy(ModuleAlarmInfo->ErrorModulePath, ModuleInfoBuffer->ModuleInformation[pModuleInfo->ModuleNumber].ModulePath);
					strcpy(ModuleAlarmInfo->ErrorModuleName, ModuleInfoBuffer->ModuleInformation[pModuleInfo->ModuleNumber].ModuleName);
					AlarmMessage = 1;
				}
				/* if various-module-plugged alarmbit is set --> reset */
				else if(ModuleAlarmInfo->AlarmBitField[pModuleInfo->ModuleNumber + OFFSET_VARIOUS_MODULE_PLUGGED] == 1)
				{	/* copy information for textsnippets */
					strcpy(ModuleAlarmInfo->ErrorModulePath, ModuleInfoBuffer->ModuleInformation[pModuleInfo->ModuleNumber].ModulePath);
					strcpy(ModuleAlarmInfo->ErrorModuleName, ModuleInfoBuffer->ModuleInformation[pModuleInfo->ModuleNumber].ErrorModuleName);
					AlarmMessage = 1;
				}
			}
			/* various module is plugged */
			else if(pModuleInfo->ActualModuleInformation.ModuleState == VAR_MODULE_PLUGGED)
			{	/* reset other alarmbits */
				if(ModuleAlarmInfo->AlarmBitField[pModuleInfo->ModuleNumber + OFFSET_MODULE_ONLY_CONFIGURED] == 1)
				{	/* copy information for textsnippets */
					strcpy(ModuleAlarmInfo->ErrorModulePath, ModuleInfoBuffer->ModuleInformation[pModuleInfo->ModuleNumber].ModulePath);
					strcpy(ModuleAlarmInfo->ErrorModuleName, ModuleInfoBuffer->ModuleInformation[pModuleInfo->ModuleNumber].ErrorModuleName);
					AlarmMessage = 1;
				}
				else if(ModuleAlarmInfo->AlarmBitField[pModuleInfo->ModuleNumber + OFFSET_MODULE_ONLY_INSERTED] == 1)
				{	/* copy information for textsnippets */
					strcpy(ModuleAlarmInfo->ErrorModulePath, ModuleInfoBuffer->ModuleInformation[pModuleInfo->ModuleNumber].ModulePath);
					strcpy(ModuleAlarmInfo->ErrorModuleName, ModuleInfoBuffer->ModuleInformation[pModuleInfo->ModuleNumber].ModuleName);
					AlarmMessage = 1;
				}
			}

			if(AlarmMessage == 0)
			{	pModuleInfo->Step = CHECK_NEW_ALARMMESSAGES;
			}
			else
			{	AlarmMessage = 0;
				pModuleInfo->LastStep = CHECK_OLD_MODULE_ALARMS;
				pModuleInfo->Step = WAIT;
			}
		break;

		/* reset module alarms */
		case RESET_MODULE_ALARMS2:
			if(pModuleInfo->ActualModuleInformation.ModuleState == MODULE_ONLY_CONFIGURED)
			{	/* reset other alarmbits */
				if(ModuleAlarmInfo->AlarmBitField[pModuleInfo->ModuleNumber + OFFSET_MODULE_ONLY_INSERTED] == 1)
				{	/* reset alarm */
					ModuleAlarmInfo->AlarmBitField[pModuleInfo->ModuleNumber + OFFSET_MODULE_ONLY_INSERTED] = 0;
				}
				else if(ModuleAlarmInfo->AlarmBitField[pModuleInfo->ModuleNumber + OFFSET_VARIOUS_MODULE_PLUGGED] == 1)
				{	/* reset alarm */
					ModuleAlarmInfo->AlarmBitField[pModuleInfo->ModuleNumber + OFFSET_VARIOUS_MODULE_PLUGGED] = 0;
				}
			}
			/* module is only inserted --> module only inserted */
			else if(pModuleInfo->ActualModuleInformation.ModuleState == MODULE_ONLY_INSERTED)
			{	/* reset other alarmbits */
				if(ModuleAlarmInfo->AlarmBitField[pModuleInfo->ModuleNumber + OFFSET_MODULE_ONLY_CONFIGURED] == 1)
				{	/* reset alarm */
					ModuleAlarmInfo->AlarmBitField[pModuleInfo->ModuleNumber + OFFSET_MODULE_ONLY_CONFIGURED] = 0;
				}
				else if(ModuleAlarmInfo->AlarmBitField[pModuleInfo->ModuleNumber + OFFSET_VARIOUS_MODULE_PLUGGED] == 1)
				{	/* reset alarm */
					ModuleAlarmInfo->AlarmBitField[pModuleInfo->ModuleNumber + OFFSET_VARIOUS_MODULE_PLUGGED] = 0;
				}
			}
			/* modulestate is OK */
			else if(pModuleInfo->ActualModuleInformation.ModuleState == MODULE_OK)
			{	/* if module-only-configured alarmbit is set --> reset */
				if(ModuleAlarmInfo->AlarmBitField[pModuleInfo->ModuleNumber + OFFSET_MODULE_ONLY_CONFIGURED] == 1)
				{	/* reset alarm */
					ModuleAlarmInfo->AlarmBitField[pModuleInfo->ModuleNumber + OFFSET_MODULE_ONLY_CONFIGURED] = 0;
				}
				/* if module-only-inserted alarmbit is set --> reset */
				else if(ModuleAlarmInfo->AlarmBitField[pModuleInfo->ModuleNumber + OFFSET_MODULE_ONLY_INSERTED] == 1)
				{	/* reset alarm */
					ModuleAlarmInfo->AlarmBitField[pModuleInfo->ModuleNumber + OFFSET_MODULE_ONLY_INSERTED] = 0;
				}
				/* if various-module-plugged alarmbit is set --> reset */
				else if(ModuleAlarmInfo->AlarmBitField[pModuleInfo->ModuleNumber + OFFSET_VARIOUS_MODULE_PLUGGED] == 1)
				{	/* reset alarm */
					ModuleAlarmInfo->AlarmBitField[pModuleInfo->ModuleNumber + OFFSET_VARIOUS_MODULE_PLUGGED] = 0;
				}
			}
			/* various module is plugged */
			else if(pModuleInfo->ActualModuleInformation.ModuleState == VAR_MODULE_PLUGGED)
			{	/* reset other alarmbits */
				if(ModuleAlarmInfo->AlarmBitField[pModuleInfo->ModuleNumber + OFFSET_MODULE_ONLY_CONFIGURED] == 1)
				{	/* reset alarm */
					ModuleAlarmInfo->AlarmBitField[pModuleInfo->ModuleNumber + OFFSET_MODULE_ONLY_CONFIGURED] = 0;
				}
				else if(ModuleAlarmInfo->AlarmBitField[pModuleInfo->ModuleNumber + OFFSET_MODULE_ONLY_INSERTED] == 1)
				{	/* reset alarm */
					ModuleAlarmInfo->AlarmBitField[pModuleInfo->ModuleNumber + OFFSET_MODULE_ONLY_INSERTED] = 0;
				}
			}
			pModuleInfo->LastStep = RESET_MODULE_ALARMS2;
			pModuleInfo->Step = WAIT;
		break;

		/* check new module alarms */
		case CHECK_NEW_ALARMMESSAGES:
			if(pModuleInfo->ActualModuleInformation.ModuleState == MODULE_ONLY_CONFIGURED)
			{	/* check alarmbit */
				if(ModuleAlarmInfo->AlarmBitField[pModuleInfo->ModuleNumber + OFFSET_MODULE_ONLY_CONFIGURED] == 0)
				{	/* copy information for textsnippets */
					strcpy(ModuleAlarmInfo->ErrorModulePath, pModuleInfo->ActualModuleInformation.ModulePath);
					strcpy(ModuleAlarmInfo->ErrorModuleName, pModuleInfo->ActualModuleInformation.ErrorModuleName);
					AlarmMessage = 1;
				}
			}
			/* module is only inserted --> module only inserted */
			else if(pModuleInfo->ActualModuleInformation.ModuleState == MODULE_ONLY_INSERTED)
			{	/* check alarmbit */
				if(ModuleAlarmInfo->AlarmBitField[pModuleInfo->ModuleNumber + OFFSET_MODULE_ONLY_INSERTED] == 0)
				{	/* copy information for textsnippets */
					strcpy(ModuleAlarmInfo->ErrorModulePath, pModuleInfo->ActualModuleInformation.ModulePath);
					strcpy(ModuleAlarmInfo->ErrorModuleName, pModuleInfo->ActualModuleInformation.ModuleName);
					AlarmMessage = 1;
				}
			}
			/* various module is plugged */
			else if(pModuleInfo->ActualModuleInformation.ModuleState == VAR_MODULE_PLUGGED)
			{	/* check alarmbit */
				if(ModuleAlarmInfo->AlarmBitField[pModuleInfo->ModuleNumber + OFFSET_VARIOUS_MODULE_PLUGGED] == 0)
				{	/* copy information for textsnippets */
					strcpy(ModuleAlarmInfo->ErrorModulePath, pModuleInfo->ActualModuleInformation.ModulePath);
					strcpy(ModuleAlarmInfo->ErrorModuleName, pModuleInfo->ActualModuleInformation.ErrorModuleName);
					AlarmMessage = 1;
				}
			}

			if(AlarmMessage == 0)
			{	pModuleInfo->Step = CHECK_NEXT_MODULE;
				/* copy data to module-buffer */
				memcpy(&(ModuleInfoBuffer->ModuleInformation[pModuleInfo->ModuleNumber]), &(pModuleInfo->ActualModuleInformation), sizeof(pModuleInfo->ActualModuleInformation));

				memset(&(pModuleInfo->ActualModuleInformation), 0, sizeof(pModuleInfo->ActualModuleInformation));

				/* next module-information */
				pModuleInfo->ModuleNumber++;
			}
			else
			{	AlarmMessage = 0;
				pModuleInfo->LastStep = CHECK_NEW_ALARMMESSAGES;
				pModuleInfo->Step = WAIT;
			}
		break;

		case SET_ALARMMESSAGES:
			if(pModuleInfo->ActualModuleInformation.ModuleState == MODULE_ONLY_CONFIGURED)
			{	/* set alarm */
				ModuleAlarmInfo->AlarmBitField[pModuleInfo->ModuleNumber + OFFSET_MODULE_ONLY_CONFIGURED] = 1;
			}
			/* module is only inserted --> module only inserted */
			else if(pModuleInfo->ActualModuleInformation.ModuleState == MODULE_ONLY_INSERTED)
			{	/* set alarm */
				ModuleAlarmInfo->AlarmBitField[pModuleInfo->ModuleNumber + OFFSET_MODULE_ONLY_INSERTED] = 1;
			}
			/* various module is plugged */
			else if(pModuleInfo->ActualModuleInformation.ModuleState == VAR_MODULE_PLUGGED)
			{	/* copy information for textsnippets */
				ModuleAlarmInfo->AlarmBitField[pModuleInfo->ModuleNumber + OFFSET_VARIOUS_MODULE_PLUGGED] = 1;
			}

			/* copy data to module-buffer */
			memcpy(&(ModuleInfoBuffer->ModuleInformation[pModuleInfo->ModuleNumber]), &(pModuleInfo->ActualModuleInformation), sizeof(pModuleInfo->ActualModuleInformation));

			memset(&(pModuleInfo->ActualModuleInformation), 0, sizeof(pModuleInfo->ActualModuleInformation));

			/* next module-information */
			pModuleInfo->ModuleNumber++;

			pModuleInfo->LastStep = SET_ALARMMESSAGES;
			pModuleInfo->Step = WAIT;
		break;

		/* next module, only 100 modules are supported */
		case CHECK_NEXT_MODULE:
			if(pModuleInfo->ModuleIndex < pModuleInfo->NumberOfTotalModules - 1)
			{	if((pModuleInfo->ModuleIndex - pModuleInfo->NumberNotCheckedModules) == MAX_MODULE_NUMBER - 1)
				{	pModuleInfo->NumberOfTotalModules = MAX_MODULE_NUMBER;
					pModuleInfo->Step = CHECK_MODULENUMBER;
				}
				else
				{	/* next module */
					pModuleInfo->ModuleIndex++;
					pModuleInfo->Step = CHECK_MODULESTATE;
				}
			}
			else
			{	pModuleInfo->Step = CHECK_MODULENUMBER;
			}
		break;

		/* check module-number */
		case CHECK_MODULENUMBER:
			if((pModuleInfo->NumberOfTotalModules - pModuleInfo->NumberNotCheckedModules) < pModuleInfo->ModulesLastCheck)
			{	pModuleInfo->ModuleDifference = pModuleInfo->ModulesLastCheck - (pModuleInfo->NumberOfTotalModules - pModuleInfo->NumberNotCheckedModules);
				pModuleInfo->Step = CHECK_NOT_NEEDED_ALARMS;
			}
			else
			{	pModuleInfo->ModulesLastCheck = (pModuleInfo->NumberOfTotalModules - pModuleInfo->NumberNotCheckedModules);
				pModuleInfo->Step = DISPOSE_INFO;
			}
		break;

		/* check not needed alarms */
		case CHECK_NOT_NEEDED_ALARMS:
			/* reset alarmbit and moduleinformationbuffer */
			if(ModuleAlarmInfo->AlarmBitField[pModuleInfo->ModuleNumber + pModuleInfo->ResetModuleAlarms + OFFSET_MODULE_ONLY_CONFIGURED] == 1)
			{	/* copy information for textsnippets */
				strcpy(ModuleAlarmInfo->ErrorModulePath, ModuleInfoBuffer->ModuleInformation[pModuleInfo->ModuleNumber + pModuleInfo->ResetModuleAlarms].ModulePath);
				strcpy(ModuleAlarmInfo->ErrorModuleName, ModuleInfoBuffer->ModuleInformation[pModuleInfo->ModuleNumber + pModuleInfo->ResetModuleAlarms].ErrorModuleName);
			}
			else if(ModuleAlarmInfo->AlarmBitField[pModuleInfo->ModuleNumber + pModuleInfo->ResetModuleAlarms + OFFSET_MODULE_ONLY_INSERTED] == 1)
			{	/* copy information for textsnippets */
				strcpy(ModuleAlarmInfo->ErrorModulePath, ModuleInfoBuffer->ModuleInformation[pModuleInfo->ModuleNumber + pModuleInfo->ResetModuleAlarms].ModulePath);
				strcpy(ModuleAlarmInfo->ErrorModuleName, ModuleInfoBuffer->ModuleInformation[pModuleInfo->ModuleNumber + pModuleInfo->ResetModuleAlarms].ModuleName);
			}
			else if(ModuleAlarmInfo->AlarmBitField[pModuleInfo->ModuleNumber + pModuleInfo->ResetModuleAlarms + OFFSET_VARIOUS_MODULE_PLUGGED] == 1)
			{	/* copy information for textsnippets */
				strcpy(ModuleAlarmInfo->ErrorModulePath, ModuleInfoBuffer->ModuleInformation[pModuleInfo->ModuleNumber + pModuleInfo->ResetModuleAlarms].ModulePath);
				strcpy(ModuleAlarmInfo->ErrorModuleName, ModuleInfoBuffer->ModuleInformation[pModuleInfo->ModuleNumber + pModuleInfo->ResetModuleAlarms].ErrorModuleName);
			}

			pModuleInfo->LastStep = CHECK_NOT_NEEDED_ALARMS;
			pModuleInfo->Step = WAIT;
		break;

		/* reset alarms */
		case RESET_NOT_NEEDED_ALARMS:
			/* reset alarmbit and moduleinformationbuffer */
			if(ModuleAlarmInfo->AlarmBitField[pModuleInfo->ModuleNumber + pModuleInfo->ResetModuleAlarms + OFFSET_MODULE_ONLY_CONFIGURED] == 1)
			{	/* reset alarm */
				ModuleAlarmInfo->AlarmBitField[pModuleInfo->ModuleNumber + pModuleInfo->ResetModuleAlarms + OFFSET_MODULE_ONLY_CONFIGURED] = 0;
			}
			else if(ModuleAlarmInfo->AlarmBitField[pModuleInfo->ModuleNumber + pModuleInfo->ResetModuleAlarms + OFFSET_MODULE_ONLY_INSERTED] == 1)
			{	/* reset alarm */
				ModuleAlarmInfo->AlarmBitField[pModuleInfo->ModuleNumber + pModuleInfo->ResetModuleAlarms + OFFSET_MODULE_ONLY_INSERTED] = 0;
			}
			else if(ModuleAlarmInfo->AlarmBitField[pModuleInfo->ModuleNumber + pModuleInfo->ResetModuleAlarms + OFFSET_VARIOUS_MODULE_PLUGGED] == 1)
			{	/* reset alarm */
				ModuleAlarmInfo->AlarmBitField[pModuleInfo->ModuleNumber + pModuleInfo->ResetModuleAlarms + OFFSET_VARIOUS_MODULE_PLUGGED] = 0;
			}

			/* reset module-buffer */
			strcpy(ModuleInfoBuffer->ModuleInformation[pModuleInfo->ModuleNumber + pModuleInfo->ResetModuleAlarms].ModuleName, "");
			strcpy(ModuleInfoBuffer->ModuleInformation[pModuleInfo->ModuleNumber + pModuleInfo->ResetModuleAlarms].ModulePath, "");
			strcpy(ModuleInfoBuffer->ModuleInformation[pModuleInfo->ModuleNumber + pModuleInfo->ResetModuleAlarms].ErrorModuleName, "");
			ModuleInfoBuffer->ModuleInformation[pModuleInfo->ModuleNumber + pModuleInfo->ResetModuleAlarms].ModuleState = 0;
			ModuleInfoBuffer->ModuleInformation[pModuleInfo->ModuleNumber + pModuleInfo->ResetModuleAlarms].ModuleColor = 0;
			strcpy(pModuleInfo->PathBuffer[pModuleInfo->ModuleNumber + pModuleInfo->ResetModuleAlarms], "");

			pModuleInfo->LastStep = RESET_NOT_NEEDED_ALARMS;
			pModuleInfo->Step = WAIT;
		break;

		/* check if other modules can be reset */
		case CHECK_RESET_NEXT_MODULE:
			if(pModuleInfo->ResetModuleAlarms < pModuleInfo->ModuleDifference - 1)
			{	pModuleInfo->ResetModuleAlarms++;
				pModuleInfo->Step = CHECK_NOT_NEEDED_ALARMS;
			}
			else
			{	pModuleInfo->ResetModuleAlarms = 0;
				pModuleInfo->ModuleDifference = 0;
				pModuleInfo->ModulesLastCheck = pModuleInfo->NumberOfTotalModules;
				pModuleInfo->Step = DISPOSE_INFO;
			}
		break;

		/* dispose HW-info */
		case DISPOSE_INFO:
			DisposeInfo.enable = 1;
			DisposeInfo.ident = CreateHWInfo.ident;

			DiagDisposeInfo(&DisposeInfo);

			if(DisposeInfo.status == 0)
			{	strcpy(ModuleAlarmInfo->ErrorModulePath, "");
				strcpy(ModuleAlarmInfo->ErrorModuleName , "");
				pModuleInfo->ModuleNumber = 0;
				pModuleInfo->status = 0;
				pModuleInfo->Step = CREATE_HW_INFO;
			}
			else if(DisposeInfo.status != 65535)
			{	pModuleInfo->status = DisposeInfo.status;
			}
		break;

		/* wait */
		case WAIT:
			pModuleInfo->WaitTimer.IN = 1;
			pModuleInfo->WaitTimer.PT = 5; /*750*/

			TON(&pModuleInfo->WaitTimer);

			if(pModuleInfo->WaitTimer.Q == 1)
			{	pModuleInfo->WaitTimer.IN = 0;
				TON(&pModuleInfo->WaitTimer);

				if(pModuleInfo->LastStep == CHECK_OLD_MODULE_PATH)
					pModuleInfo->Step = RESET_MODULE_ALARMS1;
				else if(pModuleInfo->LastStep == RESET_MODULE_ALARMS1)
				{	strcpy(ModuleAlarmInfo->ErrorModulePath, "");
					strcpy(ModuleAlarmInfo->ErrorModuleName , "");
					pModuleInfo->Step = CHECK_OLD_MODULE_ALARMS;
				}
				else if(pModuleInfo->LastStep == CHECK_OLD_MODULE_ALARMS)
					pModuleInfo->Step = RESET_MODULE_ALARMS2;
				else if(pModuleInfo->LastStep == RESET_MODULE_ALARMS2)
				{	strcpy(ModuleAlarmInfo->ErrorModulePath, "");
					strcpy(ModuleAlarmInfo->ErrorModuleName , "");
					pModuleInfo->Step = CHECK_NEW_ALARMMESSAGES;
				}
				else if(pModuleInfo->LastStep == CHECK_NEW_ALARMMESSAGES)
					pModuleInfo->Step = SET_ALARMMESSAGES;
				else if(pModuleInfo->LastStep == SET_ALARMMESSAGES)
				{	strcpy(ModuleAlarmInfo->ErrorModulePath, "");
					strcpy(ModuleAlarmInfo->ErrorModuleName , "");
					pModuleInfo->Step = CHECK_NEXT_MODULE;
				}
				else if(pModuleInfo->LastStep == CHECK_NOT_NEEDED_ALARMS)
					pModuleInfo->Step = RESET_NOT_NEEDED_ALARMS;
				else if(pModuleInfo->LastStep == RESET_NOT_NEEDED_ALARMS)
				{	strcpy(ModuleAlarmInfo->ErrorModulePath, "");
					strcpy(ModuleAlarmInfo->ErrorModuleName , "");
					pModuleInfo->Step = CHECK_RESET_NEXT_MODULE;
				}

				pModuleInfo->LastStep = 0;
			}
		break;
	}
}
```

### Program Logical/HmiHandling/HmiIO/HmiIO (IEC) - IO Handling

#### HmiIOCtrl.st - Implementation code
```iecst
(********************************************************************
 * COPYRIGHT --
 ********************************************************************
 * PROGRAM: HmiIOCtrl
 * File: HmiIOCtrl.st
 * Author: renj
 * Created: October 15, 2014
 ********************************************************************
 * Implementation OF PROGRAM HmiIOCtrl
 ********************************************************************)

PROGRAM _INIT

(* init program *)

	StatusIOList := IOList(ADR(pIOInformation));
	IOReadIndex := 0;
	MAX_IO_LINES_MINUS_ONE;
	MAX_LINES_MINUS_ONE;

	DI1;
	DI2;
	DI3;
	DI4;
	DI5;

	DO1;
	DO2;
	DO3;
	DO4;
	DO5;

END_PROGRAM

PROGRAM _CYCLIC

	ModuleDiagnose_1.AdrModuleInformationBuffer := ADR(ModuleInformation);
	ModuleDiagnose_1.Option := DiagnoseOption;
	ModuleDiagnose_1.AdrAlarmInformation := ADR(AlarmInformation);
	ModuleDiagnose_1();

	IF ModuleDiagnose_1.status = 0 THEN
		NumberOfTotalModules := ModuleDiagnose_1.NumberOfTotalModules - ModuleDiagnose_1.NumberNotCheckedModules;
		HmiIOCtrl.Output.Status.DiagnosticsInitDone := TRUE;
	END_IF

	Status := IOStatus(pIOInformation.StartAdrBuffer, ADR(pStatusBuffer), Elements, ADR(pEnableForce), ADR(pForceValue));

	pIOData ACCESS pIOInformation.StartAdrBuffer + (IOReadIndex * SIZEOF(pIOData));
	Elements := pIOInformation.TotalIONumber;

	IF  (ModuleInformation[0].ModuleName = '1A4600.10') OR
		(ModuleInformation[0].ModuleName = '1A4600.10-2') OR
		(ModuleInformation[0].ModuleName = '5PC810.SX01-00-AR010') OR
		(ModuleInformation[0].ModuleName = '5PC810.SX02-00-AR010') OR
		(ModuleInformation[0].ModuleName = '5PC810.SX05-00-AR010') OR
		(ModuleInformation[0].ModuleName = '5PC820.SX01-00-AR010') OR
		(ModuleInformation[0].ModuleName = '5PC820.SX01-01-AR010') OR
		(ModuleInformation[0].ModuleName = '1A4000.00') (*OR
		(ModuleInformation[0].ModuleName = 'X20CP1484-1') *)THEN

		HmiIOCtrl.Output.Status.SimulationActive := TRUE;

	ELSE

		HmiIOCtrl.Output.Status.SimulationActive := FALSE;

	END_IF

	IF HmiGlobal.PageControl.ActPage = PAGE_SERVICE_DIAGNOSTICS THEN

		DiagRTInfo.enable := 1;
		DiagRTInfo();

		cycT := DiagRTInfo.cycle_time / 1000;

		CASE Step OF

			INIT:

				(* Initialize the list of modules *)
				HmiIOCtrl.Output.Status.ModuleInfoLayerStatus := 0;
				HmiIOCtrl.Output.Status.IOInfoLayerStatus := 1;

				brsmemset(ADR(HmiIOCtrl.Output.ModuleInfo), 0, SIZEOF(HmiIOCtrl.Output.ModuleInfo));

				IF NumberOfTotalModules > MAX_LINES THEN
					EndIndex := MAX_LINES-1;
				ELSIF NumberOfTotalModules <= MAX_LINES AND NumberOfTotalModules > 0 THEN
					EndIndex := NumberOfTotalModules-1;
				ELSIF NumberOfTotalModules = 0 THEN
					EndIndex := 0;
				END_IF

				FOR Index := 0 TO EndIndex DO

					brsmemcpy(ADR(HmiIOCtrl.Output.ModuleInfo.ModuleName[Index]), ADR(ModuleInformation[Index].ModuleName), SIZEOF(HmiIOCtrl.Output.ModuleInfo.ModuleName[Index]));
					brsmemcpy(ADR(HmiIOCtrl.Output.ModuleInfo.ModulePath[Index]), ADR(ModuleInformation[Index].ModulePath), SIZEOF(HmiIOCtrl.Output.ModuleInfo.ModulePath[Index]));
					brsmemcpy(ADR(HmiIOCtrl.Output.ModuleInfo.ErrorModuleName[Index]), ADR(ModuleInformation[Index].ErrorModuleName), SIZEOF(HmiIOCtrl.Output.ModuleInfo.ErrorModuleName[Index]));

					HmiIOCtrl.Output.ModuleInfo.ModuleState[Index] := ModuleInformation[Index].ModuleState;

					IF (HmiIOCtrl.Output.ModuleInfo.ModuleState[Index] = 4) THEN
						HmiIOCtrl.Output.ModuleInfo.WrongModulStatus[Index] := 0;
					ELSE
						HmiIOCtrl.Output.ModuleInfo.WrongModulStatus[Index] := 1;
					END_IF

				END_FOR

				(* Color data point for the cursor of the module list*)
				ColorOld := WHITE;
				HmiIOCtrl.Output.ModuleInfo.Color[0] := ORANGE;

				SelectedIndex := 0;
				SelectedModuleIndex := 0;

				FOR Index:= 2 TO (MAX_LINES-1) BY 2 DO
					HmiIOCtrl.Output.ModuleInfo.Color[Index] := WHITE;
				END_FOR

				FOR Index := 1 TO (MAX_LINES-1) BY 2 DO
					HmiIOCtrl.Output.ModuleInfo.Color[Index] := GREY;
				END_FOR

				StartIndex:= 0;
				(* I/O layer invisible at startup*)
				HmiIOCtrl.Output.Status.StatusLayerMessage := 1;

				Step:= COMMAND;

			COMMAND:

				(** Wait for commands set from the visualization ****)
				IF NumberOfTotalModules <> NumberOfTotalModulesOld THEN
					NumberOfTotalModulesOld := NumberOfTotalModules;
					Step := INIT;
				END_IF

				HmiIOCtrl.Output.Status.PageFocusColor := BLACK_WHITE;

				IF HmiIOCtrl.Input.Command.InfoLineDown > Internal.OldCommand.InfoLineDown THEN
					IF (SelectedIndex < (MAX_LINES-1)) AND (SelectedIndex < (NumberOfTotalModules-1)) AND (NumberOfTotalModules > 0) THEN

						HmiIOCtrl.Output.ModuleInfo.Color[SelectedIndex] := ColorOld;
						SelectedIndex := SelectedIndex +1;
						SelectedModuleIndex := SelectedModuleIndex + 1;
						ColorOld := HmiIOCtrl.Output.ModuleInfo.Color[SelectedIndex];
						HmiIOCtrl.Output.ModuleInfo.Color[SelectedIndex] := ORANGE;

					ELSIF (SelectedModuleIndex < (NumberOfTotalModules-1)) AND (SelectedIndex >= (MAX_LINES-1)) THEN

						SelectedModuleIndex := SelectedModuleIndex + 1;
						StartIndex := SelectedModuleIndex-MAX_LINES+1;
						EndIndex := StartIndex+MAX_LINES-1;
						IF (EndIndex > (NumberOfTotalModules-1)) THEN
							EndIndex := NumberOfTotalModules-1;
						END_IF

						Step := UPDATE_LIST;

					END_IF

				ELSIF HmiIOCtrl.Input.Command.InfoLineUp > Internal.OldCommand.InfoLineUp THEN

					IF (SelectedIndex = 0) AND (SelectedModuleIndex > 0) THEN

						SelectedModuleIndex := SelectedModuleIndex - 1;
						StartIndex := SelectedModuleIndex;
						EndIndex := SelectedModuleIndex+MAX_LINES-1;
						Step := UPDATE_LIST;

					ELSIF (SelectedIndex > 0) THEN

						HmiIOCtrl.Output.ModuleInfo.Color[SelectedIndex] := ColorOld;
						SelectedIndex := SelectedIndex - 1;
						SelectedModuleIndex := SelectedModuleIndex - 1;
						ColorOld := HmiIOCtrl.Output.ModuleInfo.Color[SelectedIndex];
						HmiIOCtrl.Output.ModuleInfo.Color[SelectedIndex] := ORANGE;

					END_IF
					(* Update all lists after 1s*)
				ELSIF (UpdateCounter <= 1000) THEN
					UpdateCounter := UpdateCounter + cycT;
				ELSIF (UpdateCounter > 1000) THEN
					UpdateCounter := 0;
					Step := UPDATE_LIST;
				END_IF

				(* The I/O layer is displayed if I/Os are configured on this module, otherwise a warning will be displayed*)
				IF HmiIOCtrl.Input.Command.Enter > Internal.OldCommand.Enter THEN
					DetailsAvailable := 0;
					IF (pIOInformation.StartAdrBuffer <> 0) THEN
						EndValue := UINT_TO_USINT(pIOInformation.TotalIONumber)-1;
						FOR IOStartIndex := 0 TO EndValue DO
							IOReadIndex := IOStartIndex;
							pIOData ACCESS pIOInformation.StartAdrBuffer + (IOReadIndex * SIZEOF(pIOData));
							Equal := brsstrcmp(ADR(ModuleInformation[SelectedModuleIndex].ModulePath), ADR(pIOData.Device));
							IF (Equal = 0) THEN
								DetailsAvailable := 1;
								HmiIOCtrl.Output.Status.ModuleInfoLayerStatus := 1;
								HmiIOCtrl.Output.Status.IOInfoLayerStatus := 0;

								EXIT;

							END_IF
						END_FOR
						Step := IO_INIT;

					ELSE
						HmiIOCtrl.Output.Status.StatusLayerMessage := 0;
						Step:= WAIT_FOR_ACKNOWLEDGE;
					END_IF
				END_IF

			WAIT_FOR_ACKNOWLEDGE:

				IF HmiIOCtrl.Input.Command.DiscardChange > Internal.OldCommand.DiscardChange THEN

					HmiIOCtrl.Output.Status.StatusLayerMessage := 1;
					Step := COMMAND;

				END_IF

			UPDATE_LIST:

				(* Update the list of modules*)
				LineIndex:= 0;

				FOR Index:= StartIndex TO EndIndex DO
					brsmemcpy(ADR(HmiIOCtrl.Output.ModuleInfo.ModuleName[LineIndex]), ADR(ModuleInformation[Index].ModuleName), SIZEOF(HmiIOCtrl.Output.ModuleInfo.ModuleName[LineIndex]));
					brsmemcpy(ADR(HmiIOCtrl.Output.ModuleInfo.ModulePath[LineIndex]), ADR(ModuleInformation[Index].ModulePath), SIZEOF(HmiIOCtrl.Output.ModuleInfo.ModulePath[LineIndex]));
					brsmemcpy(ADR(HmiIOCtrl.Output.ModuleInfo.ErrorModuleName[LineIndex]), ADR(ModuleInformation[Index].ErrorModuleName), SIZEOF(HmiIOCtrl.Output.ModuleInfo.ErrorModuleName[LineIndex]));
					HmiIOCtrl.Output.ModuleInfo.ModuleState[LineIndex] := ModuleInformation[Index].ModuleState;
					IF (HmiIOCtrl.Output.ModuleInfo.ModuleState[LineIndex] = 4) THEN
						HmiIOCtrl.Output.ModuleInfo.WrongModulStatus[LineIndex] := 0;
					ELSE
						HmiIOCtrl.Output.ModuleInfo.WrongModulStatus[LineIndex] := 1;
					END_IF
					LineIndex := LineIndex + 1;
				END_FOR

				Step := COMMAND;

			(********************************************************************************************************************************************************)
			(*							IO Handling Layer																											*)
			(********************************************************************************************************************************************************)

			IO_INIT:

				(*Initialize the I/O list*)
				brsmemset(ADR(HmiIOCtrl.Output.IOInfo), 0, SIZEOF(HmiIOCtrl.Output.IOInfo));
				brsmemset(ADR(IOIndexArray), 0, SIZEOF(IOIndexArray));
				NumberIO := 0;
				EndValue := UINT_TO_USINT(pIOInformation.TotalIONumber)-1;

				LineIndex := 0;
				FOR Index := IOStartIndex TO EndValue DO
					IOReadIndex := Index;
					pIOData ACCESS pIOInformation.StartAdrBuffer + (IOReadIndex * SIZEOF(pIOData));
					Equal := brsstrcmp(ADR(ModuleInformation[SelectedModuleIndex].ModulePath), ADR(pIOData.Device));
					IF (Equal = 0) THEN
						IF (LineIndex < MAX_IO_LINES) THEN
							brsmemcpy(ADR(HmiIOCtrl.Output.IOInfo.PVName[LineIndex]), ADR(pIOData.PVName), SIZEOF(HmiIOCtrl.Output.IOInfo.PVName[LineIndex]));
							brsmemcpy(ADR(HmiIOCtrl.Output.IOInfo.LogicalName[LineIndex]), ADR(pIOData.LogicalName), SIZEOF(HmiIOCtrl.Output.IOInfo.LogicalName[LineIndex]));
							HmiIOCtrl.Output.IOInfo.DiagnosicsType[LineIndex] := pStatusBuffer[Index].DataType;
							HmiIOCtrl.Output.IOInfo.ActValue[LineIndex] := pStatusBuffer[Index].ActValue;
							HmiIOCtrl.Output.IOInfo.ForceValue[LineIndex] := pForceValue[Index];
							HmiIOCtrl.Output.IOInfo.EnableForcing[LineIndex] := pEnableForce[Index];
							HmiIOCtrl.Output.IOInfo.InivisibleLines[LineIndex] := 0;
							IOIndexArray[LineIndex] := Index;
							(* Set min and max value of the numeric input fields *)
							CASE HmiIOCtrl.Output.IOInfo.DiagnosicsType[LineIndex] OF

								1:(*BOOL*)
									HmiIOCtrl.Output.IOInfo.MinValue[LineIndex] := MIN_VALUE_BOOL;
									HmiIOCtrl.Output.IOInfo.MaxValue[LineIndex] := MAX_VALUE_BOOL;

								2:(*SINT*)
									HmiIOCtrl.Output.IOInfo.MinValue[LineIndex] := MIN_VALUE_SINT;
									HmiIOCtrl.Output.IOInfo.MaxValue[LineIndex] := MAX_VALUE_SINT;

								3:(*INT*)
									HmiIOCtrl.Output.IOInfo.MinValue[LineIndex] := MIN_VALUE_INT;
									HmiIOCtrl.Output.IOInfo.MaxValue[LineIndex] := MAX_VALUE_INT;

								4:(*DINT*)
									HmiIOCtrl.Output.IOInfo.MinValue[LineIndex] := MIN_VALUE_DINT;
									HmiIOCtrl.Output.IOInfo.MaxValue[LineIndex] := MAX_VALUE_DINT;

								5:(*USINT*)
									HmiIOCtrl.Output.IOInfo.MinValue[LineIndex] := MIN_VALUE_USINT;
									HmiIOCtrl.Output.IOInfo.MaxValue[LineIndex] := MAX_VALUE_USINT;

								6:(*UINT*)
									HmiIOCtrl.Output.IOInfo.MinValue[LineIndex] := MIN_VALUE_UINT;
									HmiIOCtrl.Output.IOInfo.MaxValue[LineIndex] := MAX_VALUE_UINT;

								7:(*UDINT*)
									HmiIOCtrl.Output.IOInfo.MinValue[LineIndex] := MIN_VALUE_UDINT;
									HmiIOCtrl.Output.IOInfo.MaxValue[LineIndex] := MAX_VALUE_UDINT;

							END_CASE

							LineIndex := LineIndex+1;

						END_IF

						NumberIO := NumberIO+1;

					ELSE
						EXIT;
					END_IF
				END_FOR

				brsmemcpy(ADR(HmiIOCtrl.Output.IOInfo.ModuleName), ADR(ModuleInformation[SelectedModuleIndex].ModuleName), SIZEOF(HmiIOCtrl.Output.IOInfo.ModuleName));
				brsmemcpy(ADR(HmiIOCtrl.Output.IOInfo.ModulePath), ADR(ModuleInformation[SelectedModuleIndex].ModulePath), SIZEOF(HmiIOCtrl.Output.IOInfo.ModulePath));
				HmiIOCtrl.Output.IOInfo.ModuleStatus := ModuleInformation[SelectedModuleIndex].ModuleState;

				IF (LineIndex < (MAX_IO_LINES-1)) THEN
					FOR InvisibleIndex := LineIndex TO (MAX_IO_LINES-1) DO
						HmiIOCtrl.Output.IOInfo.InivisibleLines[InvisibleIndex]:= 1;
					END_FOR
				END_IF

				(*Color of the cursor of the I/O list*)
				ColorOld := WHITE;
				ColorNumericOld := NUMERIC_WHITE;
				HmiIOCtrl.Output.IOInfo.Color[0] := ORANGE;
				HmiIOCtrl.Output.IOInfo.NumericColor[0] := NUMERIC_ORANGE;
				SelectedLineIndex := 0;
				SelectedIOIndex := IOStartIndex;
				FOR Index:= 2 TO (MAX_IO_LINES-1) BY 2 DO
					HmiIOCtrl.Output.IOInfo.Color[Index] := WHITE;
					HmiIOCtrl.Output.IOInfo.NumericColor[Index] := NUMERIC_WHITE;
				END_FOR

				FOR Index:= 1 TO (MAX_IO_LINES-1) BY 2 DO
					HmiIOCtrl.Output.IOInfo.Color[Index] := GREY;
					HmiIOCtrl.Output.IOInfo.NumericColor[Index] := NUMERIC_GREY;
				END_FOR

				HmiIOCtrl.Output.Status.IOInfoLayerStatus := 0;
				HmiIOCtrl.Output.Status.ModuleInfoLayerStatus := 1;
				StartIndex := IOStartIndex;
				IF (NumberIO = 1) THEN
					EndIndex := StartIndex;
				ELSIF (NumberIO < MAX_IO_LINES-1) THEN
					EndIndex:= IOStartIndex+NumberIO-1;
				ELSE
					EndIndex:= StartIndex+MAX_IO_LINES-1;
				END_IF

				HmiIOCtrl.Output.Status.StatusLayerMessage := 1;

				pv_adr := 0;
				Step := IO_GETADDR;

			IO_GETADDR:

				IF (EndIndex>StartIndex) AND (StartIndex<pIOInformation.TotalIONumber) THEN

					status_adr := PV_xgetadr(ADR(HmiIOCtrl.Output.IOInfo.PVName[0]), ADR(pv_adr), ADR(data_len));

					IF 	status_adr = 0 AND pv_adr <> 0 THEN

						HmiIOCtrl.Output.IOInfo.SelectedIO.ForceValue := HmiIOCtrl.Output.IOInfo.ForceValue[0];
						brsmemcpy(ADR(HmiIOCtrl.Output.IOInfo.SelectedIO.LogicalName), ADR(HmiIOCtrl.Output.IOInfo.LogicalName[0]), SIZEOF(HmiIOCtrl.Output.IOInfo.SelectedIO.LogicalName));
						brsmemcpy(ADR(HmiIOCtrl.Output.IOInfo.SelectedIO.PVName), ADR(HmiIOCtrl.Output.IOInfo.PVName[0]), SIZEOF(HmiIOCtrl.Output.IOInfo.SelectedIO.PVName));
						HmiIOCtrl.Output.IOInfo.SelectedIO.MinValue := HmiIOCtrl.Output.IOInfo.MinValue[0];
						HmiIOCtrl.Output.IOInfo.SelectedIO.MaxValue := HmiIOCtrl.Output.IOInfo.MaxValue[0];

						Step := IO_COMMAND;

					END_IF

				ELSE

					HmiIOCtrl.Output.IOInfo.SelectedIO.ForceValue := HmiIOCtrl.Output.IOInfo.ForceValue[0];
					brsmemcpy(ADR(HmiIOCtrl.Output.IOInfo.SelectedIO.LogicalName), ADR(HmiIOCtrl.Output.IOInfo.LogicalName[0]), SIZEOF(HmiIOCtrl.Output.IOInfo.SelectedIO.LogicalName));
					brsmemcpy(ADR(HmiIOCtrl.Output.IOInfo.SelectedIO.PVName), ADR(HmiIOCtrl.Output.IOInfo.PVName[0]), SIZEOF(HmiIOCtrl.Output.IOInfo.SelectedIO.PVName));
					HmiIOCtrl.Output.IOInfo.SelectedIO.MinValue := HmiIOCtrl.Output.IOInfo.MinValue[0];
					HmiIOCtrl.Output.IOInfo.SelectedIO.MaxValue := HmiIOCtrl.Output.IOInfo.MaxValue[0];

					Step := IO_COMMAND;

				END_IF

			IO_COMMAND:

				IF HmiIOCtrl.Input.Command.DiscardChange > Internal.OldCommand.DiscardChange THEN

					HmiIOCtrl.Output.Status.ModuleInfoLayerStatus := 0;
					HmiIOCtrl.Output.Status.IOInfoLayerStatus := 1;
					Step := INIT;

				ELSIF HmiIOCtrl.Input.Command.ForcingOn > Internal.OldCommand.ForcingOn THEN

					HmiIOCtrl.Output.IOInfo.EnableForcing[SelectedLineIndex] := 1;
					pEnableForce[SelectedIOIndex] := 1;
					HmiIOCtrl.Output.Status.IOForced := 0;

					FOR ResetIndex:= 0 TO (UINT_TO_USINT(Elements)-1) DO
						IF (pEnableForce[ResetIndex] = 1)THEN
							HmiIOCtrl.Output.Status.IOForced := 1;
						END_IF
					END_FOR

					Step := ENABLE_FORCE;

				ELSIF HmiIOCtrl.Input.Command.ForcingOff > Internal.OldCommand.ForcingOff THEN

					HmiIOCtrl.Output.IOInfo.EnableForcing[SelectedLineIndex] := 0;
					pEnableForce[SelectedIOIndex] := 0;
					HmiIOCtrl.Output.Status.IOForced := 0;

					FOR ResetIndex:= 0 TO (UINT_TO_USINT(Elements)-1) DO
						IF (pEnableForce[ResetIndex] = 1)THEN
							HmiIOCtrl.Output.Status.IOForced := 1;
						END_IF
					END_FOR

					Step:= DISABLE_FORCE;

				ELSIF HmiIOCtrl.Input.Command.ForcingAllOff > Internal.OldCommand.ForcingAllOff THEN

					FOR ResetIndex := 0 TO (UINT_TO_USINT(Elements)-1) DO
						pEnableForce[ResetIndex]:= 0;
					END_FOR
					HmiIOCtrl.Output.Status.IOForced := 0;
					Step := UPDATE_IO_LIST;

				ELSIF HmiIOCtrl.Input.Command.InfoLineDown > Internal.OldCommand.InfoLineDown THEN

					IF (SelectedLineIndex < (MAX_IO_LINES-1)) AND (SelectedLineIndex < (NumberIO-1)) AND (NumberIO > 0) THEN

						HmiIOCtrl.Output.IOInfo.Color[SelectedLineIndex] := ColorOld;
						HmiIOCtrl.Output.IOInfo.NumericColor[SelectedLineIndex] := ColorNumericOld;
						SelectedLineIndex := SelectedLineIndex +1;
						SelectedIOIndex := SelectedIOIndex + 1;
						ColorOld := HmiIOCtrl.Output.IOInfo.Color[SelectedLineIndex];
						HmiIOCtrl.Output.IOInfo.Color[SelectedLineIndex] := ORANGE;
						ColorNumericOld := HmiIOCtrl.Output.IOInfo.NumericColor[SelectedLineIndex];
						HmiIOCtrl.Output.IOInfo.NumericColor[SelectedLineIndex] := NUMERIC_ORANGE;

					ELSIF ((SelectedIOIndex-StartIndex) < (NumberIO-1)) AND (SelectedLineIndex >= (MAX_IO_LINES-1)) THEN

						IF ((SelectedIOIndex-IOStartIndex) < (NumberIO-1)) THEN
							SelectedIOIndex := SelectedIOIndex + 1;
							StartIndex := SelectedIOIndex-MAX_IO_LINES+1;
							EndIndex := StartIndex+MAX_IO_LINES-1;
							IF (EndIndex > (NumberIO-1+IOStartIndex)) THEN
								EndIndex := NumberIO-1;
							END_IF

							Step := UPDATE_IO_LIST;

						END_IF

					END_IF

					HmiIOCtrl.Output.IOInfo.SelectedIO.ForceValue := HmiIOCtrl.Output.IOInfo.ForceValue[SelectedLineIndex];
					brsmemcpy(ADR(HmiIOCtrl.Output.IOInfo.SelectedIO.LogicalName), ADR(HmiIOCtrl.Output.IOInfo.LogicalName[SelectedLineIndex]), SIZEOF(HmiIOCtrl.Output.IOInfo.SelectedIO.LogicalName));
					brsmemcpy(ADR(HmiIOCtrl.Output.IOInfo.SelectedIO.PVName), ADR(HmiIOCtrl.Output.IOInfo.PVName[SelectedLineIndex]), SIZEOF(HmiIOCtrl.Output.IOInfo.SelectedIO.PVName));
					HmiIOCtrl.Output.IOInfo.SelectedIO.MinValue := HmiIOCtrl.Output.IOInfo.MinValue[SelectedLineIndex];
					HmiIOCtrl.Output.IOInfo.SelectedIO.MaxValue := HmiIOCtrl.Output.IOInfo.MaxValue[SelectedLineIndex];

				ELSIF HmiIOCtrl.Input.Command.InfoLineUp > Internal.OldCommand.InfoLineUp THEN

					IF (SelectedLineIndex = 0) AND (SelectedIOIndex > IOStartIndex) THEN

						SelectedIOIndex := SelectedIOIndex - 1;
						StartIndex := SelectedIOIndex;
						EndIndex := SelectedIOIndex+MAX_IO_LINES-1;
						Step:= UPDATE_IO_LIST;

					ELSIF (SelectedLineIndex > 0) THEN

						HmiIOCtrl.Output.IOInfo.Color[SelectedLineIndex] := ColorOld;
						HmiIOCtrl.Output.IOInfo.NumericColor[SelectedLineIndex] := ColorNumericOld;
						SelectedLineIndex := SelectedLineIndex - 1;
						SelectedIOIndex := SelectedIOIndex - 1;
						ColorOld := HmiIOCtrl.Output.IOInfo.Color[SelectedLineIndex];
						HmiIOCtrl.Output.IOInfo.Color[SelectedLineIndex] := ORANGE;
						ColorNumericOld := HmiIOCtrl.Output.IOInfo.NumericColor[SelectedLineIndex];
						HmiIOCtrl.Output.IOInfo.NumericColor[SelectedLineIndex] := NUMERIC_ORANGE;

					END_IF

					HmiIOCtrl.Output.IOInfo.SelectedIO.ForceValue := HmiIOCtrl.Output.IOInfo.ForceValue[SelectedLineIndex];
					brsmemcpy(ADR(HmiIOCtrl.Output.IOInfo.SelectedIO.LogicalName), ADR(HmiIOCtrl.Output.IOInfo.LogicalName[SelectedLineIndex]), SIZEOF(HmiIOCtrl.Output.IOInfo.SelectedIO.LogicalName));
					brsmemcpy(ADR(HmiIOCtrl.Output.IOInfo.SelectedIO.PVName), ADR(HmiIOCtrl.Output.IOInfo.PVName[SelectedLineIndex]), SIZEOF(HmiIOCtrl.Output.IOInfo.SelectedIO.PVName));
					HmiIOCtrl.Output.IOInfo.SelectedIO.MinValue := HmiIOCtrl.Output.IOInfo.MinValue[SelectedLineIndex];
					HmiIOCtrl.Output.IOInfo.SelectedIO.MaxValue := HmiIOCtrl.Output.IOInfo.MaxValue[SelectedLineIndex];

				ELSIF HmiIOCtrl.Input.Command.PageDown > Internal.OldCommand.PageDown THEN

					FOR Index := SelectedModuleIndex+1 TO NumberOfTotalModules-1 DO

						IF (brsstrcmp(ADR(ModuleInformation[Index].ModuleName), ADR('X20DI9371')) = 0) OR
							(brsstrcmp(ADR(ModuleInformation[Index].ModuleName), ADR('X20DO9322')) = 0) THEN

							SelectedModuleIndex :=Index;
							Step := PAGE_CHANGE;

							EXIT;
						END_IF

					END_FOR

				ELSIF HmiIOCtrl.Input.Command.PageUp > Internal.OldCommand.PageUp THEN

					FOR Index := SelectedModuleIndex-1 TO 1 BY -1 DO

						IF (brsstrcmp(ADR(ModuleInformation[Index].ModuleName), ADR('X20DI9371')) = 0) OR
							(brsstrcmp(ADR(ModuleInformation[Index].ModuleName), ADR('X20DO9322')) = 0) THEN

							SelectedModuleIndex := Index;
							Step := PAGE_CHANGE;

							EXIT;
						END_IF
					END_FOR

				ELSIF HmiIOCtrl.Input.Command.SetValue THEN

					HmiIOCtrl.Input.Command.SetValue := 0;

					HmiIOCtrl.Output.IOInfo.ForceValue[SelectedLineIndex] := HmiIOCtrl.Output.IOInfo.SelectedIO.ForceValue;
					pForceValue[SelectedIOIndex] := HmiIOCtrl.Output.IOInfo.SelectedIO.ForceValue;

					IF (HmiIOCtrl.Output.IOInfo.EnableForcing[SelectedLineIndex] = 1) THEN
						Step := UPDATE_FORCE_VALUE;
					END_IF

				ELSIF (UpdateIOCounter <= 1000) THEN
					UpdateIOCounter := UpdateIOCounter + cycT;
				ELSIF (UpdateIOCounter > 1000) THEN
					UpdateIOCounter := 0;
					Step := UPDATE_IO_LIST;
				END_IF

				HmiIOCtrl.Output.IOInfo.ModuleStatus := ModuleInformation[SelectedModuleIndex].ModuleState;

			ENABLE_FORCE:

				IF (HmiIOCtrl.Output.IOInfo.EnableForcing[SelectedLineIndex] = 1) THEN

					IF (brsstrcmp(ADR(ModuleInformation[SelectedModuleIndex].ModuleName), ADR('X20DI9371')) = 0) THEN
						brsstrcpy(ADR(PointData),ADR('%IX.'));
					ELSIF (brsstrcmp(ADR(ModuleInformation[SelectedModuleIndex].ModuleName), ADR('X20DO9322')) = 0) THEN
						brsstrcpy(ADR(PointData),ADR('%QX.'));
					END_IF

					brsstrcat(ADR(PointData), ADR(HmiIOCtrl.Output.IOInfo.ModulePath));
					brsstrcat(ADR(PointData), ADR('.'));
					brsstrcat(ADR(PointData), ADR(HmiIOCtrl.Output.IOInfo.LogicalName[SelectedLineIndex]));

					IODPEnableForce.enable := 1;
					IODPEnableForce.pDatapoint := ADR(PointData);

					IODPEnableForce();

					IF(IODPEnableForce.status = 0)THEN
						Step := UPDATE_FORCE_VALUE;
					ELSIF(IODPEnableForce.status <> 65535) THEN
						Step := IO_COMMAND;
					END_IF
				ELSE
					Step := IO_COMMAND;
				END_IF

			DISABLE_FORCE:

				IF (brsstrcmp(ADR(ModuleInformation[SelectedModuleIndex].ModuleName), ADR('X20DI9371')) = 0)THEN
					brsstrcpy(ADR(PointData), ADR('%IX.'));
				ELSIF (brsstrcmp(ADR(ModuleInformation[SelectedModuleIndex].ModuleName),ADR('X20DO9322')) = 0)THEN
					brsstrcpy(ADR(PointData), ADR('%QX.'));
				END_IF

				brsstrcat(ADR(PointData), ADR(HmiIOCtrl.Output.IOInfo.ModulePath));
				brsstrcat(ADR(PointData), ADR('.'));
				brsstrcat(ADR(PointData), ADR(HmiIOCtrl.Output.IOInfo.LogicalName[SelectedLineIndex]));

				IODPDisableForce.enable := 1;

				IODPDisableForce.pDatapoint :=  ADR(PointData);

				IODPDisableForce();

				IF(IODPDisableForce.status = 0)	THEN
					Step := IO_COMMAND;
				ELSIF (IODPDisableForce.status <> 65535)THEN
					Step := IO_COMMAND;
				END_IF

			UPDATE_FORCE_VALUE:

				IF (HmiIOCtrl.Output.IOInfo.EnableForcing[SelectedLineIndex]=1)THEN

					IF (brsstrcmp(ADR(ModuleInformation[SelectedModuleIndex].ModuleName), ADR('X20DI9371')) = 0) THEN
						brsstrcpy(ADR(PointData), ADR('%IX.'));
					ELSIF (brsstrcmp(ADR(ModuleInformation[SelectedModuleIndex].ModuleName),ADR('X20DO9322')) = 0) THEN
						brsstrcpy(ADR(PointData), ADR('%QX.'));
					END_IF

					brsstrcat(ADR(PointData), ADR(HmiIOCtrl.Output.IOInfo.ModulePath));
					brsstrcat(ADR(PointData), ADR('.'));
					brsstrcat(ADR(PointData), ADR(HmiIOCtrl.Output.IOInfo.LogicalName[SelectedLineIndex]));

					IODPSetForceValue.enable := 1;

					IODPSetForceValue.pDatapoint :=  ADR(PointData);

					IODPSetForceValue.value := pForceValue[SelectedIOIndex];

					IODPSetForceValue();

					IF(IODPSetForceValue.status = 0)THEN
						Step := IO_COMMAND;
					ELSIF(IODPSetForceValue.status <> 65535) THEN
						Step := IO_COMMAND;
					END_IF
				ELSE
					Step := IO_COMMAND;
				END_IF

			PAGE_CHANGE:

				DetailsAvailable := 0;

				IF (pIOInformation.StartAdrBuffer <> 0) THEN

					EndValue := UINT_TO_USINT(pIOInformation.TotalIONumber)-1;

					FOR IOStartIndex := 0 TO EndValue DO

						IOReadIndex := IOStartIndex;
						pIOData ACCESS pIOInformation.StartAdrBuffer + (IOReadIndex * SIZEOF(pIOData));
						Equal := brsstrcmp(ADR(ModuleInformation[SelectedModuleIndex].ModulePath), ADR(pIOData.Device));

						IF (Equal = 0) THEN

							DetailsAvailable := 1;
							HmiIOCtrl.Output.Status.ModuleInfoLayerStatus := 1;
							HmiIOCtrl.Output.Status.IOInfoLayerStatus := 0;
							Step := IO_INIT;
							EXIT;

						ELSE

							Step := IO_INIT;

						END_IF

					END_FOR

				ELSE

					Step := IO_INIT;

				END_IF

			CHANGE_FORCE_VALUE:

				HmiIOCtrl.Output.IOInfo.SelectedIO.Status := 0;

				HmiIOCtrl.Output.Status.PageFocusColor := WHITE_ORANGE;;

				IF HmiIOCtrl.Input.Command.SetValue THEN

					HmiIOCtrl.Input.Command.SetValue := 0;

					HmiIOCtrl.Output.IOInfo.ForceValue[SelectedLineIndex] := HmiIOCtrl.Output.IOInfo.SelectedIO.ForceValue;
					HmiIOCtrl.Output.IOInfo.SelectedIO.Status := 2;
					pForceValue[SelectedIOIndex] := HmiIOCtrl.Output.IOInfo.SelectedIO.ForceValue;

					Step := IO_COMMAND;

				ELSIF HmiIOCtrl.Input.Command.DiscardChange > Internal.OldCommand.DiscardChange THEN

					HmiIOCtrl.Output.IOInfo.SelectedIO.Status := 2;

					Step:= IO_COMMAND;

				END_IF

			UPDATE_IO_LIST:

				(*Update the I/O list entries*)
				LineIndex := 0;

				FOR Index := StartIndex TO EndIndex DO

					IOReadIndex := Index;
					pIOData ACCESS pIOInformation.StartAdrBuffer + (IOReadIndex * SIZEOF(pIOData));
					brsmemcpy(ADR(HmiIOCtrl.Output.IOInfo.PVName[LineIndex]), ADR(pIOData.PVName), SIZEOF(HmiIOCtrl.Output.IOInfo.PVName[LineIndex]));
					brsmemcpy(ADR(HmiIOCtrl.Output.IOInfo.LogicalName[LineIndex]), ADR(pIOData.LogicalName), SIZEOF(HmiIOCtrl.Output.IOInfo.LogicalName[LineIndex]));

					HmiIOCtrl.Output.IOInfo.DiagnosicsType[LineIndex] := pStatusBuffer[Index].DataType;
					HmiIOCtrl.Output.IOInfo.ActValue[LineIndex] := pStatusBuffer[Index].ActValue;
					HmiIOCtrl.Output.IOInfo.ForceValue[LineIndex] := pForceValue[Index];
					HmiIOCtrl.Output.IOInfo.EnableForcing[LineIndex] := pEnableForce[Index];
					HmiIOCtrl.Output.IOInfo.InivisibleLines[LineIndex] := 0;
					IOIndexArray[LineIndex] := Index;

					CASE HmiIOCtrl.Output.IOInfo.DiagnosicsType[LineIndex] OF

						1:(*BOOL*)
							HmiIOCtrl.Output.IOInfo.MinValue[LineIndex] := MIN_VALUE_BOOL;
							HmiIOCtrl.Output.IOInfo.MaxValue[LineIndex] := MAX_VALUE_BOOL;

						2:(*SINT*)
							HmiIOCtrl.Output.IOInfo.MinValue[LineIndex] := MIN_VALUE_SINT;
							HmiIOCtrl.Output.IOInfo.MaxValue[LineIndex] := MAX_VALUE_SINT;

						3:(*INT*)
							HmiIOCtrl.Output.IOInfo.MinValue[LineIndex] := MIN_VALUE_INT;
							HmiIOCtrl.Output.IOInfo.MaxValue[LineIndex] := MAX_VALUE_INT;

						4:(*DINT*)
							HmiIOCtrl.Output.IOInfo.MinValue[LineIndex] := MIN_VALUE_DINT;
							HmiIOCtrl.Output.IOInfo.MaxValue[LineIndex] := MAX_VALUE_DINT;

						5:(*USINT*)
							HmiIOCtrl.Output.IOInfo.MinValue[LineIndex] := MIN_VALUE_USINT;
							HmiIOCtrl.Output.IOInfo.MaxValue[LineIndex] := MAX_VALUE_USINT;

						6:(*UINT*)
							HmiIOCtrl.Output.IOInfo.MinValue[LineIndex] := MIN_VALUE_UINT;
							HmiIOCtrl.Output.IOInfo.MaxValue[LineIndex] := MAX_VALUE_UINT;

						7:(*UDINT*)
							HmiIOCtrl.Output.IOInfo.MinValue[LineIndex] := MIN_VALUE_UDINT;
							HmiIOCtrl.Output.IOInfo.MaxValue[LineIndex] := MAX_VALUE_UDINT;

					END_CASE

					LineIndex := LineIndex + 1;

				END_FOR

				HmiIOCtrl.Output.IOInfo.SelectedIO.ForceValue := HmiIOCtrl.Output.IOInfo.ForceValue[SelectedLineIndex];
				brsmemcpy(ADR(HmiIOCtrl.Output.IOInfo.SelectedIO.LogicalName), ADR(HmiIOCtrl.Output.IOInfo.LogicalName[SelectedLineIndex]), SIZEOF(HmiIOCtrl.Output.IOInfo.SelectedIO.LogicalName));
				brsmemcpy(ADR(HmiIOCtrl.Output.IOInfo.SelectedIO.PVName), ADR(HmiIOCtrl.Output.IOInfo.PVName[SelectedLineIndex]), SIZEOF(HmiIOCtrl.Output.IOInfo.SelectedIO.PVName));
				HmiIOCtrl.Output.IOInfo.SelectedIO.MinValue := HmiIOCtrl.Output.IOInfo.MinValue[SelectedLineIndex];
				HmiIOCtrl.Output.IOInfo.SelectedIO.MaxValue := HmiIOCtrl.Output.IOInfo.MaxValue[SelectedLineIndex];

				Step := IO_COMMAND;

		END_CASE

		IF (HmiIOCtrl.Output.Status.IOInfoLayerStatus = 0) THEN
			HmiIOCtrl.Output.Status.IOInformationStatus := 1;
		ELSE
			HmiIOCtrl.Output.Status.IOInformationStatus := 0;
		END_IF

	ELSE	(*Other page*)

		Step := INIT;

	END_IF

	Internal.OldCommand := HmiIOCtrl.Input.Command;

END_PROGRAM
```

#### HmiIOCtrlLocal.typ - Local data types
```iecst
(********************************************************************
 * COPYRIGHT --
 ********************************************************************
 * Program: HmiIOCtrl
 * File: HmiIOCtrlLocal.typ
 * Author: renj
 * Created: October 15, 2014
 ********************************************************************
 * Local data types of program HmiIOCtrl
 ********************************************************************)

TYPE
	HmiIOCtrlInternal_Type : 	STRUCT
		OldCommand : HmiIOCtrlInputCommand_Type;
	END_STRUCT;
END_TYPE
```

#### HmiIOCtrlLocal.var - Local variables
```iecst
(********************************************************************
 * COPYRIGHT --
 ********************************************************************
 * Program: HmiIOCtrl
 * File: HmiIOCtrlLocal.var
 * Author: renj
 * Created: October 15, 2014
 ********************************************************************
 * Local variables of program HmiIOCtrl
 ********************************************************************)
VAR CONSTANT
	BLACK_WHITE : UINT := 15;
	WHITE_ORANGE : UINT := 4093;
	CHANGE_FORCE_VALUE : USINT := 6;
	COMMAND : USINT := 1;
	MAX_VALUE_BOOL : BOOL := 1;
	MAX_VALUE_DINT : DINT := 2147483647;
	MAX_VALUE_INT : INT := 32767;
	MAX_VALUE_SINT : SINT := 127;
	MAX_VALUE_UDINT : UDINT := 4294967295;
	MAX_VALUE_UINT : UINT := 65535;
	MAX_VALUE_USINT : USINT := 255;
	MIN_VALUE_BOOL : BOOL := 0;
	MIN_VALUE_DINT : DINT := -2147483648;
	MIN_VALUE_INT : INT := -32768;
	MIN_VALUE_SINT : SINT := -128;
	MIN_VALUE_UDINT : UDINT := 0;
	MIN_VALUE_UINT : UINT := 0;
	MIN_VALUE_USINT : USINT := 0;
	GREY : UINT := 63738;
	INIT : USINT := 0;
	IO_COMMAND : USINT := 4;
	IO_INIT : USINT := 3;
	NUMERIC_GREY : UINT := 250;
	NUMERIC_ORANGE : UINT := 253;
	NUMERIC_WHITE : UINT := 15;
	ORANGE : UINT := 63741;
	PAGE_SERVICE_DIAGNOSTICS : UINT := 300;
	UPDATE_IO_LIST : USINT := 5;
	UPDATE_LIST : USINT := 2;
	WHITE : UINT := 63503;
	WAIT_FOR_ACKNOWLEDGE : USINT := 17;
	PAGE_CHANGE : USINT := 20;
	IO_GETADDR : USINT := 15;
	UPDATE_FORCE_VALUE : USINT := 32;
	ENABLE_FORCE : USINT := 30;
	DISABLE_FORCE : USINT := 31;
END_VAR
VAR
	AlarmInformation : ModuleAlarmInformation_typ;
	ColorNumericOld : UINT;
	ColorOld : UINT;
	DetailsAvailable : BOOL;
	DiagnoseOption : USINT;
	Elements : UINT;
	EndIndex : USINT;
	EndValue : USINT;
	Equal : DINT;
	Index : USINT;
	InvisibleIndex : USINT;
	IOIndexArray : ARRAY[0..MAX_IO_LINES_MINUS_ONE] OF USINT;
	IOReadIndex : USINT;
	IOStartIndex : USINT;
	LineIndex : USINT;
	ModuleDiagnose_1 : ModuleDiagnose;
	ModuleInformation : ARRAY[0..99] OF ModuleInformation_Type;
	NumberIO : USINT;
	NumberOfTotalModules : USINT;
	NumberOfTotalModulesOld : USINT;
	pEnableForce : ARRAY[0..254] OF BOOL;
	pForceValue : ARRAY[0..254] OF DINT;
	pIOData : REFERENCE TO SingleIOEntry_typ;
	pIOInformation : IODPList_typ;
	pStatusBuffer : ARRAY[0..254] OF SingleIOStatus_typ;
	ResetIndex : USINT;
	SelectedIndex : USINT;
	SelectedIOIndex : USINT;
	SelectedLineIndex : USINT;
	SelectedModuleIndex : USINT;
	StartIndex : USINT;
	Status : UINT;
	StatusIOList : UINT;
	Step : USINT;
	UpdateCounter : UDINT;
	status_adr : UINT;
	pv_adr : UDINT;
	data_len : UDINT;
	PointData : STRING[60];
	IODPEnableForce : AsIOEnableForcing;
	IODPDisableForce : AsIODisableForcing;
	IODPSetForceValue : AsIOSetForceValue;
	Internal : HmiIOCtrlInternal_Type := (0);
	DiagRTInfo : RTInfo;
	cycT : UDINT;
	UpdateIOCounter : UDINT;
END_VAR
```

### Package Logical/HmiHandling/HmiPrg - Prg Manage Page

### HmiProgramGlobal.typ - Global data types
```iecst
(********************************************************************
 * COPYRIGHT -- Bernecker + Rainer
 ********************************************************************
 * Program: HmiProgram
 * File: HmiProgramInterface.typ
 * Author: B&R, International Applications
 * Created: October 08, 2008
 ********************************************************************
 * Local data types of program HmiProgram
 ********************************************************************)

TYPE
	HmiProgramLayerDefaultType : 	STRUCT
		Layer : HmiLayerType;
		ListboxFiles : HmiListboxType;
		ListboxDevices : HmiListboxType;
		ButtonPageDown : HmiButtonType;
		ButtonPageUp : HmiButtonType;
		ButtonRename : HmiButtonType;
		ButtonEdit : HmiButtonType;
		ButtonLoad : HmiButtonType;
		ButtonNew : HmiButtonType;
		ButtonDelete : HmiButtonType;
		ButtonPaste : HmiButtonType;
		ButtonCopy : HmiButtonType;
		ButtonCut : HmiButtonType;
		ScaleScrollbar : HmiScaleType;
	END_STRUCT;
	HmiProgramComponentsType : 	STRUCT
		LayerDefault : HmiProgramLayerDefaultType;
		LayerDeletePopup : HmiPopupType;
		LayerNewPopup : HmiPopupWithStringType;
		LayerRenamePopup : HmiPopupWithStringType;
		LayerCutPopup : HmiPopupType;
	END_STRUCT;
	HmiProgram_Type : 	STRUCT
		Components : HmiProgramComponentsType;
	END_STRUCT;
END_TYPE
```

### HmiProgramGlobal.var - Global variables
```iecst
(********************************************************************
 * COPYRIGHT --
 ********************************************************************
 * Package: HmiProgram
 * File: HmiProgramGlobal.var
 * Author: renj
 * Created: July 30, 2014
 ********************************************************************
 * Variables of package HmiProgram
 ********************************************************************)
VAR
	HmiProgram : HmiProgram_Type := (0);
END_VAR
```

### Program Logical/HmiHandling/HmiPrg/HmiPrg (ANSIC) - File Manager
